LIN {X 0,Y 73.269,Z 1097.58,A -85,B 0,C 180,E1 32760.013,E2 32760.013} C_VEL
LIN {X 0,Y 72.331,Z 1070.54,A -85,B 0,C 180,E1 32774.928,E2 32774.928} C_VEL
LIN {X 0,Y 74.049,Z 1040.132,A -85,B 0,C 180,E1 32785.713,E2 32785.713} C_VEL
LIN {X 0,Y 75.716,Z 1012.125,A -85,B 0,C 180,E1 32791.765,E2 32791.765} C_VEL
LIN {X 0,Y 78.944,Z 1000.666,A -85,B 0,C 180,E1 32799.89,E2 32799.89} C_VEL
LIN {X 0,Y 85.957,Z 982.06,A -85,B 0,C 180,E1 32811.287,E2 32811.287} C_VEL
LIN {X 0,Y 92.075,Z 967.893,A -85,B 0,C 180,E1 32817.665,E2 32817.665} C_VEL
LIN {X 0,Y 97.491,Z 977.138,A -85,B 0,C 180,E1 32834.538,E2 32834.538} C_VEL
LIN {X 0,Y 99.424,Z 982.889,A -85,B 0,C 180,E1 32839.493,E2 32839.493} C_VEL
LIN {X 0,Y 102.891,Z 1004.981,A -85,B 0,C 180,E1 32851.504,E2 32851.504} C_VEL
LIN {X 0,Y 105.917,Z 1033.576,A -85,B 0,C 180,E1 32864.114,E2 32864.114} C_VEL
LIN {X 0,Y 108.13,Z 1063.069,A -85,B 0,C 180,E1 32876.43,E2 32876.43} C_VEL
LIN {X 0,Y 91.376,Z 1095.603,A -85,B 0,C 180,E1 32887.248,E2 32887.248} C_VEL
LIN {X 0,Y 75.131,Z 1127.363,A -85,B 0,C 180,E1 32906.405,E2 32906.405} C_VEL
LIN {X 0,Y 68.306,Z 1151.794,A -85,B 0,C 180,E1 32932.192,E2 32932.192} C_VEL
LIN {X 0,Y 69.608,Z 1165.233,A -85,B 0,C 180,E1 32952.524,E2 32952.524} C_VEL
LIN {X 0,Y 72.852,Z 1171.689,A -85,B 0,C 180,E1 32964.037,E2 32964.037} C_VEL
LIN {X 0,Y 74.21,Z 1174.974,A -85,B 0,C 180,E1 32972.734,E2 32972.734} C_VEL
LIN {X 0,Y 75.278,Z 1177.096,A -85,B 0,C 180,E1 32981.863,E2 32981.863} C_VEL
LIN {X 0,Y 76.32,Z 1177.928,A -85,B 0,C 180,E1 32984.944,E2 32984.944} C_VEL
LIN {X 0,Y 64.876,Z 1167.053,A -85,B 0,C 180,E1 33016.653,E2 33016.653} C_VEL
LIN {X 0,Y 64.458,Z 1162.406,A -85,B 0,C 180,E1 33026.759,E2 33026.759} C_VEL
LIN {X 0,Y 69.223,Z 1138.874,A -85,B 0,C 180,E1 33059.162,E2 33059.162} C_VEL
LIN {X 0,Y 77.507,Z 1130.596,A -85,B 0,C 180,E1 33067.478,E2 33067.478} C_VEL
LIN {X 0,Y 86.454,Z 1136.917,A -85,B 0,C 180,E1 33081.75,E2 33081.75} C_VEL
LIN {X 0,Y 88.495,Z 1137.46,A -85,B 0,C 180,E1 33084.935,E2 33084.935} C_VEL
LIN {X 0,Y 71.845,Z 1114.418,A -85,B 0,C 180,E1 33102.582,E2 33102.582} C_VEL
LIN {X 0,Y 65.942,Z 1089.767,A -85,B 0,C 180,E1 33120.835,E2 33120.835} C_VEL
LIN {X 0,Y 65.245,Z 1061.691,A -85,B 0,C 180,E1 33136.079,E2 33136.079} C_VEL
LIN {X 0,Y 66.642,Z 1034.04,A -85,B 0,C 180,E1 33146.198,E2 33146.198} C_VEL
LIN {X 0,Y 68.109,Z 1027.676,A -85,B 0,C 180,E1 33151.99,E2 33151.99} C_VEL
LIN {X 0,Y 72.601,Z 1016.135,A -85,B 0,C 180,E1 33156.945,E2 33156.945} C_VEL
LIN {X 0,Y 88.946,Z 978.744,A -85,B 0,C 180,E1 33179.557,E2 33179.557} C_VEL
LIN {X 0,Y 90.136,Z 977.435,A -85,B 0,C 180,E1 33181.585,E2 33181.585} C_VEL
LIN {X 0,Y 94.291,Z 984.5,A -85,B 0,C 180,E1 33194.097,E2 33194.097} C_VEL
LIN {X 0,Y 96.446,Z 998.943,A -85,B 0,C 180,E1 33203.737,E2 33203.737} C_VEL
LIN {X 0,Y 98.608,Z 1023.035,A -85,B 0,C 180,E1 33215.969,E2 33215.969} C_VEL
LIN {X 0,Y 100.362,Z 1052.462,A -85,B 0,C 180,E1 33229.311,E2 33229.311} C_VEL
LIN {X 0,Y 100.749,Z 1064.923,A -85,B 0,C 180,E1 33234.814,E2 33234.814} C_VEL
LIN {X 0,Y 80.54,Z 1101.135,A -85,B 0,C 180,E1 33248.2,E2 33248.2} C_VEL
LIN {X 0,Y 65.83,Z 1129.761,A -85,B 0,C 180,E1 33268.887,E2 33268.887} C_VEL
LIN {X 0,Y 60.684,Z 1152.02,A -85,B 0,C 180,E1 33296.409,E2 33296.409} C_VEL
LIN {X 0,Y 63.78,Z 1165.667,A -85,B 0,C 180,E1 33320.077,E2 33320.077} C_VEL
LIN {X 0,Y 75.278,Z 1177.096,A -85,B 0,C 180,E1 33341.863,E2 33341.863} C_VEL
LIN {X 0,Y 73.492,Z 1176.552,A -85,B 0,C 180,E1 33346.07,E2 33346.07} C_VEL
LIN {X 0,Y 61.63,Z 1169.7,A -85,B 0,C 180,E1 33356.97,E2 33356.97} C_VEL
LIN {X 0,Y 57.635,Z 1160.709,A -85,B 0,C 180,E1 33382.601,E2 33382.601} C_VEL
LIN {X 0,Y 60.537,Z 1138.156,A -85,B 0,C 180,E1 33418.076,E2 33418.076} C_VEL
LIN {X 0,Y 72.588,Z 1126.229,A -85,B 0,C 180,E1 33431.005,E2 33431.005} C_VEL
LIN {X 0,Y 80.021,Z 1131.328,A -85,B 0,C 180,E1 33443.585,E2 33443.585} C_VEL
LIN {X 0,Y 64.193,Z 1107.032,A -85,B 0,C 180,E1 33462.394,E2 33462.394} C_VEL
LIN {X 0,Y 58.753,Z 1082.208,A -85,B 0,C 180,E1 33480.937,E2 33480.937} C_VEL
LIN {X 0,Y 57.93,Z 1055.888,A -85,B 0,C 180,E1 33496.145,E2 33496.145} C_VEL
LIN {X 0,Y 59.201,Z 1047.428,A -85,B 0,C 180,E1 33505.556,E2 33505.556} C_VEL
LIN {X 0,Y 62.564,Z 1038.679,A -85,B 0,C 180,E1 33510.898,E2 33510.898} C_VEL
LIN {X 0,Y 66.244,Z 1028.558,A -85,B 0,C 180,E1 33518.87,E2 33518.87} C_VEL
LIN {X 0,Y 70.701,Z 1018.492,A -85,B 0,C 180,E1 33523.474,E2 33523.474} C_VEL
LIN {X 0,Y 87.345,Z 985.981,A -85,B 0,C 180,E1 33542.477,E2 33542.477} C_VEL
LIN {X 0,Y 90.25,Z 990.494,A -85,B 0,C 180,E1 33551.862,E2 33551.862} C_VEL
LIN {X 0,Y 91.426,Z 1000.781,A -85,B 0,C 180,E1 33559.484,E2 33559.484} C_VEL
LIN {X 0,Y 92.615,Z 1023.861,A -85,B 0,C 180,E1 33572.255,E2 33572.255} C_VEL
LIN {X 0,Y 93.504,Z 1052.595,A -85,B 0,C 180,E1 33586.339,E2 33586.339} C_VEL
LIN {X 0,Y 93.778,Z 1064.964,A -85,B 0,C 180,E1 33592.325,E2 33592.325} C_VEL
LIN {X 0,Y 74.007,Z 1099.068,A -85,B 0,C 180,E1 33605.219,E2 33605.219} C_VEL
LIN {X 0,Y 57.888,Z 1128.86,A -85,B 0,C 180,E1 33628.51,E2 33628.51} C_VEL
LIN {X 0,Y 53.268,Z 1149.848,A -85,B 0,C 180,E1 33657.947,E2 33657.947} C_VEL
LIN {X 0,Y 57.119,Z 1163.179,A -85,B 0,C 180,E1 33683.362,E2 33683.362} C_VEL
LIN {X 0,Y 67.223,Z 1172.897,A -85,B 0,C 180,E1 33702.869,E2 33702.869} C_VEL
LIN {X 0,Y 67.587,Z 1173.302,A -85,B 0,C 180,E1 33705.478,E2 33705.478} C_VEL
LIN {X 0,Y 61.63,Z 1169.7,A -85,B 0,C 180,E1 33716.97,E2 33716.97} C_VEL
LIN {X 0,Y 56.714,Z 1164.958,A -85,B 0,C 180,E1 33727.877,E2 33727.877} C_VEL
LIN {X 0,Y 49.623,Z 1154.018,A -85,B 0,C 180,E1 33747.821,E2 33747.821} C_VEL
LIN {X 0,Y 55.431,Z 1132.611,A -85,B 0,C 180,E1 33783.2,E2 33783.2} C_VEL
LIN {X 0,Y 67.962,Z 1121.517,A -85,B 0,C 180,E1 33794.648,E2 33794.648} C_VEL
LIN {X 0,Y 71.157,Z 1124.078,A -85,B 0,C 180,E1 33800.442,E2 33800.442} C_VEL
LIN {X 0,Y 71.261,Z 1123.721,A -85,B 0,C 180,E1 33802.452,E2 33802.452} C_VEL
LIN {X 0,Y 56.613,Z 1098.605,A -85,B 0,C 180,E1 33822.254,E2 33822.254} C_VEL
LIN {X 0,Y 51.874,Z 1079.167,A -85,B 0,C 180,E1 33837.931,E2 33837.931} C_VEL
LIN {X 0,Y 50.419,Z 1070.196,A -85,B 0,C 180,E1 33850.815,E2 33850.815} C_VEL
LIN {X 0,Y 52.781,Z 1060.211,A -85,B 0,C 180,E1 33861.06,E2 33861.06} C_VEL
LIN {X 0,Y 56.042,Z 1049.349,A -85,B 0,C 180,E1 33872.654,E2 33872.654} C_VEL
LIN {X 0,Y 59.41,Z 1041.697,A -85,B 0,C 180,E1 33877.872,E2 33877.872} C_VEL
LIN {X 0,Y 64.941,Z 1030.146,A -85,B 0,C 180,E1 33885.654,E2 33885.654} C_VEL
LIN {X 0,Y 70.113,Z 1019.904,A -85,B 0,C 180,E1 33890.545,E2 33890.545} C_VEL
LIN {X 0,Y 85.198,Z 994.192,A -85,B 0,C 180,E1 33905.357,E2 33905.357} C_VEL
LIN {X 0,Y 86.763,Z 999.12,A -85,B 0,C 180,E1 33912.164,E2 33912.164} C_VEL
LIN {X 0,Y 87.019,Z 1019.939,A -85,B 0,C 180,E1 33925.462,E2 33925.462} C_VEL
LIN {X 0,Y 86.841,Z 1046.993,A -85,B 0,C 180,E1 33939.931,E2 33939.931} C_VEL
LIN {X 0,Y 86.732,Z 1065.405,A -85,B 0,C 180,E1 33949.592,E2 33949.592} C_VEL
LIN {X 0,Y 66.137,Z 1099.464,A -85,B 0,C 180,E1 33963.197,E2 33963.197} C_VEL
LIN {X 0,Y 49.307,Z 1129.404,A -85,B 0,C 180,E1 33990.11,E2 33990.11} C_VEL
LIN {X 0,Y 46.044,Z 1148.807,A -85,B 0,C 180,E1 34022.331,E2 34022.331} C_VEL
LIN {X 0,Y 51.733,Z 1161.812,A -85,B 0,C 180,E1 34050.132,E2 34050.132} C_VEL
LIN {X 0,Y 59.063,Z 1168.261,A -85,B 0,C 180,E1 34063.449,E2 34063.449} C_VEL
LIN {X 0,Y 55.452,Z 1166.083,A -85,B 0,C 180,E1 34073.716,E2 34073.716} C_VEL
LIN {X 0,Y 50.452,Z 1157.108,A -85,B 0,C 180,E1 34101.541,E2 34101.541} C_VEL
LIN {X 0,Y 49.623,Z 1154.018,A -85,B 0,C 180,E1 34107.821,E2 34107.821} C_VEL
LIN {X 0,Y 46.659,Z 1146.453,A -85,B 0,C 180,E1 34120.097,E2 34120.097} C_VEL
LIN {X 0,Y 45.254,Z 1133.912,A -85,B 0,C 180,E1 34139.18,E2 34139.18} C_VEL
LIN {X 0,Y 46.03,Z 1132.614,A -85,B 0,C 180,E1 34141.155,E2 34141.155} C_VEL
LIN {X 0,Y 61.583,Z 1117.997,A -85,B 0,C 180,E1 34157.58,E2 34157.58} C_VEL
LIN {X 0,Y 63.777,Z 1116.677,A -85,B 0,C 180,E1 34158.781,E2 34158.781} C_VEL
LIN {X 0,Y 64.034,Z 1116.775,A -85,B 0,C 180,E1 34160.044,E2 34160.044} C_VEL
LIN {X 0,Y 58.379,Z 1109.531,A -85,B 0,C 180,E1 34165.532,E2 34165.532} C_VEL
LIN {X 0,Y 46.971,Z 1093.398,A -85,B 0,C 180,E1 34186.84,E2 34186.84} C_VEL
LIN {X 0,Y 45.464,Z 1083.478,A -85,B 0,C 180,E1 34200.552,E2 34200.552} C_VEL
LIN {X 0,Y 45.37,Z 1072.217,A -85,B 0,C 180,E1 34218.091,E2 34218.091} C_VEL
LIN {X 0,Y 48.213,Z 1063.415,A -85,B 0,C 180,E1 34228.232,E2 34228.232} C_VEL
LIN {X 0,Y 54.1,Z 1050.421,A -85,B 0,C 180,E1 34240.916,E2 34240.916} C_VEL
LIN {X 0,Y 64.463,Z 1031.664,A -85,B 0,C 180,E1 34252.58,E2 34252.58} C_VEL
LIN {X 0,Y 70.388,Z 1021.454,A -85,B 0,C 180,E1 34257.406,E2 34257.406} C_VEL
LIN {X 0,Y 81.875,Z 1004.023,A -85,B 0,C 180,E1 34267.37,E2 34267.37} C_VEL
LIN {X 0,Y 82.7,Z 1003.402,A -85,B 0,C 180,E1 34268.468,E2 34268.468} C_VEL
LIN {X 0,Y 81.933,Z 1022.116,A -85,B 0,C 180,E1 34281.289,E2 34281.289} C_VEL
LIN {X 0,Y 80.598,Z 1048.537,A -85,B 0,C 180,E1 34296.633,E2 34296.633} C_VEL
LIN {X 0,Y 79.874,Z 1065.624,A -85,B 0,C 180,E1 34306.312,E2 34306.312} C_VEL
LIN {X 0,Y 59.759,Z 1097.562,A -85,B 0,C 180,E1 34319.305,E2 34319.305} C_VEL
LIN {X 0,Y 41.409,Z 1128.292,A -85,B 0,C 180,E1 34349.857,E2 34349.857} C_VEL
LIN {X 0,Y 39.175,Z 1147.808,A -85,B 0,C 180,E1 34388.69,E2 34388.69} C_VEL
LIN {X 0,Y 50.045,Z 1162.565,A -85,B 0,C 180,E1 34423.182,E2 34423.182} C_VEL
LIN {X 0,Y 51.23,Z 1163.45,A -85,B 0,C 180,E1 34426.003,E2 34426.003} C_VEL
LIN {X 0,Y 44.027,Z 1155.114,A -85,B 0,C 180,E1 34455.264,E2 34455.264} C_VEL
LIN {X 0,Y 41.905,Z 1141.177,A -85,B 0,C 180,E1 34485.879,E2 34485.879} C_VEL
LIN {X 0,Y 46.03,Z 1132.614,A -85,B 0,C 180,E1 34501.155,E2 34501.155} C_VEL
LIN {X 0,Y 51.776,Z 1117.439,A -85,B 0,C 180,E1 34519.22,E2 34519.22} C_VEL
LIN {X 0,Y 52.783,Z 1116.6,A -85,B 0,C 180,E1 34519.963,E2 34519.963} C_VEL
LIN {X 0,Y 52.701,Z 1114.158,A -85,B 0,C 180,E1 34522.478,E2 34522.478} C_VEL
LIN {X 0,Y 40.236,Z 1097.736,A -85,B 0,C 180,E1 34547.208,E2 34547.208} C_VEL
LIN {X 0,Y 38.845,Z 1086.815,A -85,B 0,C 180,E1 34565.605,E2 34565.605} C_VEL
LIN {X 0,Y 41.251,Z 1073.821,A -85,B 0,C 180,E1 34587.276,E2 34587.276} C_VEL
LIN {X 0,Y 51.882,Z 1053.742,A -85,B 0,C 180,E1 34608.301,E2 34608.301} C_VEL
LIN {X 0,Y 64.406,Z 1033.964,A -85,B 0,C 180,E1 34619.298,E2 34619.298} C_VEL
LIN {X 0,Y 70.085,Z 1025.154,A -85,B 0,C 180,E1 34623.161,E2 34623.161} C_VEL
LIN {X 0,Y 78.268,Z 1014.107,A -85,B 0,C 180,E1 34629.629,E2 34629.629} C_VEL
LIN {X 0,Y 75.978,Z 1036.049,A -85,B 0,C 180,E1 34644.193,E2 34644.193} C_VEL
LIN {X 0,Y 73.393,Z 1064.578,A -85,B 0,C 180,E1 34661.774,E2 34661.774} C_VEL
LIN {X 0,Y 71.768,Z 1068.969,A -85,B 0,C 180,E1 34663.684,E2 34663.684} C_VEL
LIN {X 0,Y 48.037,Z 1103.645,A -85,B 0,C 180,E1 34680.072,E2 34680.072} C_VEL
LIN {X 0,Y 32.019,Z 1131.042,A -85,B 0,C 180,E1 34717.825,E2 34717.825} C_VEL
LIN {X 0,Y 33.455,Z 1147.512,A -85,B 0,C 180,E1 34759.772,E2 34759.772} C_VEL
LIN {X 0,Y 42.399,Z 1157.413,A -85,B 0,C 180,E1 34785.432,E2 34785.432} C_VEL
LIN {X 0,Y 38.023,Z 1152.822,A -85,B 0,C 180,E1 34806.804,E2 34806.804} C_VEL
LIN {X 0,Y 34.899,Z 1145.661,A -85,B 0,C 180,E1 34827.116,E2 34827.116} C_VEL
LIN {X 0,Y 42.009,Z 1126.064,A -85,B 0,C 180,E1 34869.242,E2 34869.242} C_VEL
LIN {X 0,Y 52.783,Z 1116.6,A -85,B 0,C 180,E1 34879.963,E2 34879.963} C_VEL
LIN {X 0,Y 51.395,Z 1113.671,A -85,B 0,C 180,E1 34883.224,E2 34883.224} C_VEL
LIN {X 0,Y 36.084,Z 1107.544,A -85,B 0,C 180,E1 34896.539,E2 34896.539} C_VEL
LIN {X 0,Y 35.699,Z 1107.001,A -85,B 0,C 180,E1 34897.623,E2 34897.623} C_VEL
LIN {X 0,Y 32.687,Z 1089.505,A -85,B 0,C 180,E1 34933.845,E2 34933.845} C_VEL
LIN {X 0,Y 38.353,Z 1075.343,A -85,B 0,C 180,E1 34958.016,E2 34958.016} C_VEL
LIN {X 0,Y 50.178,Z 1057.544,A -85,B 0,C 180,E1 34975.943,E2 34975.943} C_VEL
LIN {X 0,Y 65.017,Z 1036.397,A -85,B 0,C 180,E1 34985.916,E2 34985.916} C_VEL
LIN {X 0,Y 72.206,Z 1026.65,A -85,B 0,C 180,E1 34990.403,E2 34990.403} C_VEL
LIN {X 0,Y 73.006,Z 1025.797,A -85,B 0,C 180,E1 34991.067,E2 34991.067} C_VEL
LIN {X 0,Y 69.36,Z 1048.529,A -85,B 0,C 180,E1 35006.382,E2 35006.382} C_VEL
LIN {X 0,Y 66.702,Z 1067.325,A -85,B 0,C 180,E1 35018.844,E2 35018.844} C_VEL
LIN {X 0,Y 41.562,Z 1102.19,A -85,B 0,C 180,E1 35034.586,E2 35034.586} C_VEL
LIN {X 0,Y 24.042,Z 1130.282,A -85,B 0,C 180,E1 35081.554,E2 35081.554} C_VEL
LIN {X 0,Y 28.514,Z 1146.066,A -85,B 0,C 180,E1 35131.963,E2 35131.963} C_VEL
LIN {X 0,Y 33.734,Z 1151.068,A -85,B 0,C 180,E1 35146.21,E2 35146.21} C_VEL
LIN {X 0,Y 34.262,Z 1151.479,A -85,B 0,C 180,E1 35150.343,E2 35150.343} C_VEL
LIN {X 0,Y 30.015,Z 1146.152,A -85,B 0,C 180,E1 35171.929,E2 35171.929} C_VEL
LIN {X 0,Y 34.271,Z 1123.987,A -85,B 0,C 180,E1 35231.699,E2 35231.699} C_VEL
LIN {X 0,Y 42.454,Z 1116.366,A -85,B 0,C 180,E1 35241.976,E2 35241.976} C_VEL
LIN {X 0,Y 42.067,Z 1114.607,A -85,B 0,C 180,E1 35244.351,E2 35244.351} C_VEL
LIN {X 0,Y 35.699,Z 1107.001,A -85,B 0,C 180,E1 35257.623,E2 35257.623} C_VEL
LIN {X 0,Y 28.843,Z 1098.236,A -85,B 0,C 180,E1 35282.374,E2 35282.374} C_VEL
LIN {X 0,Y 28.812,Z 1089.021,A -85,B 0,C 180,E1 35312.75,E2 35312.75} C_VEL
LIN {X 0,Y 49.374,Z 1061.151,A -85,B 0,C 180,E1 35344.074,E2 35344.074} C_VEL
LIN {X 0,Y 65.343,Z 1040.222,A -85,B 0,C 180,E1 35352.14,E2 35352.14} C_VEL
LIN {X 0,Y 66.192,Z 1038.969,A -85,B 0,C 180,E1 35352.339,E2 35352.339} C_VEL
LIN {X 0,Y 66.097,Z 1041.687,A -85,B 0,C 180,E1 35355.293,E2 35355.293} C_VEL
LIN {X 0,Y 61.079,Z 1066.087,A -85,B 0,C 180,E1 35372.663,E2 35372.663} C_VEL
LIN {X 0,Y 57.823,Z 1071.773,A -85,B 0,C 180,E1 35374.725,E2 35374.725} C_VEL
LIN {X 0,Y 32.295,Z 1104.572,A -85,B 0,C 180,E1 35390.56,E2 35390.56} C_VEL
LIN {X 0,Y 16.295,Z 1129.964,A -85,B 0,C 180,E1 35451.378,E2 35451.378} C_VEL
LIN {X 0,Y 24.296,Z 1143.57,A -85,B 0,C 180,E1 35505.714,E2 35505.714} C_VEL
LIN {X 0,Y 25.874,Z 1144.891,A -85,B 0,C 180,E1 35509.553,E2 35509.553} C_VEL
LIN {X 0,Y 25.994,Z 1144.851,A -85,B 0,C 180,E1 35514.819,E2 35514.819} C_VEL
LIN {X 0,Y 28.171,Z 1120.39,A -85,B 0,C 180,E1 35598.109,E2 35598.109} C_VEL
LIN {X 0,Y 32.174,Z 1116.859,A -85,B 0,C 180,E1 35603.711,E2 35603.711} C_VEL
LIN {X 0,Y 30.671,Z 1113.321,A -85,B 0,C 180,E1 35610.517,E2 35610.517} C_VEL
LIN {X 0,Y 27.268,Z 1092.908,A -85,B 0,C 180,E1 35663.205,E2 35663.205} C_VEL
LIN {X 0,Y 28.812,Z 1089.021,A -85,B 0,C 180,E1 35672.75,E2 35672.75} C_VEL
LIN {X 0,Y 35.544,Z 1079.445,A -85,B 0,C 180,E1 35696.596,E2 35696.596} C_VEL
LIN {X 0,Y 44.353,Z 1070.714,A -85,B 0,C 180,E1 35709.683,E2 35709.683} C_VEL
LIN {X 0,Y 45.731,Z 1069.178,A -85,B 0,C 180,E1 35710.609,E2 35710.609} C_VEL
LIN {X 0,Y 56.628,Z 1056.346,A -85,B 0,C 180,E1 35715.374,E2 35715.374} C_VEL
LIN {X 0,Y 58.863,Z 1054.447,A -85,B 0,C 180,E1 35717.251,E2 35717.251} C_VEL
LIN {X 0,Y 55.414,Z 1067.461,A -85,B 0,C 180,E1 35727.239,E2 35727.239} C_VEL
LIN {X 0,Y 31.391,Z 1097.873,A -85,B 0,C 180,E1 35736.613,E2 35736.613} C_VEL
LIN {X 0,Y 9.111,Z 1125.263,A -85,B 0,C 180,E1 35804.447,E2 35804.447} C_VEL
LIN {X 0,Y 15.122,Z 1135.696,A -85,B 0,C 180,E1 35868.451,E2 35868.451} C_VEL
LIN {X 0,Y 16.665,Z 1136.873,A -85,B 0,C 180,E1 35877.525,E2 35877.525} C_VEL
LIN {X 0,Y 22.427,Z 1116.885,A -85,B 0,C 180,E1 35967.477,E2 35967.477} C_VEL
LIN {X 0,Y 20.407,Z 1111.748,A -85,B 0,C 180,E1 35982.937,E2 35982.937} C_VEL
LIN {X 0,Y 22.626,Z 1096.332,A -85,B 0,C 180,E1 36035.81,E2 36035.81} C_VEL
LIN {X 0,Y 45.731,Z 1069.178,A -85,B 0,C 180,E1 36070.609,E2 36070.609} C_VEL
LIN {X 0,Y 44.852,Z 1072.124,A -85,B 0,C 180,E1 36074.392,E2 36074.392} C_VEL
LIN {X 0,Y 41.744,Z 1077.469,A -85,B 0,C 180,E1 36077.222,E2 36077.222} C_VEL
LIN {X 0,Y 30.68,Z 1092.541,A -85,B 0,C 180,E1 36082.761,E2 36082.761} C_VEL
LIN {X 0,Y 26.509,Z 1097.161,A -85,B 0,C 180,E1 36083.846,E2 36083.846} C_VEL
LIN {X 0,Y 2.448,Z 1123.705,A -85,B 0,C 180,E1 36216.376,E2 36216.376} C_VEL
LIN {X 0,Y 5.22,Z 1126.269,A -85,B 0,C 180,E1 36243.143,E2 36243.143} C_VEL
LIN {X 0,Y 5.976,Z 1124.362,A -85,B 0,C 180,E1 36286.527,E2 36286.527} C_VEL
LIN {X 0,Y 13.057,Z 1116.834,A -85,B 0,C 180,E1 36336.165,E2 36336.165} C_VEL
LIN {X 0,Y 13.817,Z 1107.56,A -85,B 0,C 180,E1 36384.287,E2 36384.287} C_VEL
LIN {X 0,Y 32.953,Z 1086.113,A -85,B 0,C 180,E1 36431.646,E2 36431.646} C_VEL
LIN {X 0,Y 46.159,Z 1073.026,A -85,B 0,C 180,E1 36439.252,E2 36439.252} C_VEL
LIN {X 0,Y 45.095,Z 1075.295,A -85,B 0,C 180,E1 36440.903,E2 36440.903} C_VEL
LIN {X 0,Y 26.509,Z 1097.161,A -85,B 0,C 180,E1 36443.846,E2 36443.846} C_VEL
LIN {X 0,Y 25.96,Z 1098.539,A -85,B 0,C 180,E1 36443.92,E2 36443.92} C_VEL
LIN {X 0,Y 25.96,Z 1240.5,A -85,B 0,C 180,E1 36443.92,E2 36443.92} C_VEL
LIN {X 0,Y 25.96,Z 1240.5,A -85,B 0,C 180,E1 36443.92,E2 36443.92}

QRS_NEXT_CUT()
PTP {E1 36537.196,E2 36537.196}
PTP {X 0,Y 759.917,A -85,B 0,C 180,E1 36537.196,E2 36537.196,E3 0,E4 0,E5 0,E6 0}
QRS_SPEED_INIT()
LIN {X 0,Y 759.917,Z 1240.5,A -85,B 0,C 180,E1 36537.196,E2 36537.196,E3 0,E4 0,E5 0,E6 0} C_VEL
LIN {X 0,Y 759.917,Z 1178.221,A -85,B 0,C 180,E1 36537.196,E2 36537.196} C_VEL
LIN {X 0,Y 759.917,Z 1169.947,A -85,B 0,C 180,E1 36537.196,E2 36537.196} C_VEL
LIN {X 0,Y 759.916,Z 1167.96,A -85,B 0,C 180,E1 36537.062,E2 36537.062} C_VEL
LIN {X 0,Y 759.918,Z 1164.115,A -85,B 0,C 180,E1 36535.398,E2 36535.398} C_VEL
LIN {X 0,Y 759.917,Z 1158.554,A -85,B 0,C 180,E1 36533.732,E2 36533.732} C_VEL
LIN {X 0,Y 759.907,Z 1151.554,A -85,B 0,C 180,E1 36532.137,E2 36532.137} C_VEL
LIN {X 0,Y 759.915,Z 1143.032,A -85,B 0,C 180,E1 36530.612,E2 36530.612} C_VEL
LIN {X 0,Y 759.91,Z 1132.05,A -85,B 0,C 180,E1 36528.988,E2 36528.988} C_VEL
LIN {X 0,Y 759.905,Z 1120.121,A -85,B 0,C 180,E1 36527.509,E2 36527.509} C_VEL
LIN {X 0,Y 759.908,Z 1107.146,A -85,B 0,C 180,E1 36526.146,E2 36526.146} C_VEL
LIN {X 0,Y 759.913,Z 1092.503,A -85,B 0,C 180,E1 36524.823,E2 36524.823} C_VEL
LIN {X 0,Y 759.914,Z 1075.894,A -85,B 0,C 180,E1 36523.53,E2 36523.53} C_VEL
LIN {X 0,Y 759.919,Z 1058.852,A -85,B 0,C 180,E1 36522.386,E2 36522.386} C_VEL
LIN {X 0,Y 759.915,Z 1040.391,A -85,B 0,C 180,E1 36521.329,E2 36521.329} C_VEL
LIN {X 0,Y 759.917,Z 1021.211,A -85,B 0,C 180,E1 36520.398,E2 36520.398} C_VEL
LIN {X 0,Y 759.914,Z 1000.768,A -85,B 0,C 180,E1 36519.562,E2 36519.562} C_VEL
LIN {X 0,Y 759.918,Z 980.784,A -85,B 0,C 180,E1 36518.891,E2 36518.891} C_VEL
LIN {X 0,Y 759.914,Z 960.216,A -85,B 0,C 180,E1 36518.343,E2 36518.343} C_VEL
LIN {X 0,Y 759.906,Z 939.489,A -85,B 0,C 180,E1 36517.917,E2 36517.917} C_VEL
LIN {X 0,Y 759.907,Z 918.44,A -85,B 0,C 180,E1 36517.621,E2 36517.621} C_VEL
LIN {X 0,Y 759.917,Z 637.061,A -85,B 0,C 180,E1 36514.768,E2 36514.768} C_VEL
LIN {X 0,Y 759.907,Z 623.96,A -85,B 0,C 180,E1 36514.622,E2 36514.622} C_VEL
LIN {X 0,Y 759.883,Z 606.01,A -85,B 0,C 180,E1 36513.089,E2 36513.089} C_VEL
LIN {X 0,Y 759.884,Z 606.015,A -85,B 0,C 180,E1 36510.129,E2 36510.129} C_VEL
LIN {X 0,Y 759.822,Z 606.015,A -85,B 0,C 180,E1 36507.619,E2 36507.619} C_VEL
LIN {X 0,Y 759.857,Z 606.015,A -85,B 0,C 180,E1 36505.176,E2 36505.176} C_VEL
LIN {X 0,Y 759.885,Z 606.007,A -85,B 0,C 180,E1 36502.183,E2 36502.183} C_VEL
LIN {X 0,Y 759.903,Z 606.014,A -85,B 0,C 180,E1 36499.362,E2 36499.362} C_VEL
LIN {X 0,Y 759.911,Z 606.004,A -85,B 0,C 180,E1 36496.36,E2 36496.36} C_VEL
LIN {X 0,Y 759.874,Z 606.013,A -85,B 0,C 180,E1 36493.384,E2 36493.384} C_VEL
LIN {X 0,Y 759.831,Z 606.014,A -85,B 0,C 180,E1 36490.946,E2 36490.946} C_VEL
LIN {X 0,Y 759.895,Z 606.015,A -85,B 0,C 180,E1 36488.299,E2 36488.299} C_VEL
LIN {X 0,Y 759.859,Z 606.01,A -85,B 0,C 180,E1 36485.463,E2 36485.463} C_VEL
LIN {X 0,Y 759.905,Z 606.014,A -85,B 0,C 180,E1 36482.739,E2 36482.739} C_VEL
LIN {X 0,Y 759.909,Z 606.004,A -85,B 0,C 180,E1 36479.74,E2 36479.74} C_VEL
LIN {X 0,Y 759.885,Z 606.013,A -85,B 0,C 180,E1 36476.83,E2 36476.83} C_VEL
LIN {X 0,Y 759.851,Z 606.011,A -85,B 0,C 180,E1 36474.235,E2 36474.235} C_VEL
LIN {X 0,Y 759.897,Z 606.015,A -85,B 0,C 180,E1 36471.457,E2 36471.457} C_VEL
LIN {X 0,Y 759.84,Z 606.012,A -85,B 0,C 180,E1 36468.809,E2 36468.809} C_VEL
LIN {X 0,Y 759.895,Z 606.014,A -85,B 0,C 180,E1 36466.199,E2 36466.199} C_VEL
LIN {X 0,Y 759.906,Z 606.004,A -85,B 0,C 180,E1 36463.236,E2 36463.236} C_VEL
LIN {X 0,Y 759.898,Z 606.013,A -85,B 0,C 180,E1 36460.31,E2 36460.31} C_VEL
LIN {X 0,Y 759.874,Z 606.008,A -85,B 0,C 180,E1 36457.562,E2 36457.562} C_VEL
LIN {X 0,Y 759.859,Z 606.015,A -85,B 0,C 180,E1 36454.605,E2 36454.605} C_VEL
LIN {X 0,Y 759.824,Z 606.014,A -85,B 0,C 180,E1 36452.113,E2 36452.113} C_VEL
LIN {X 0,Y 759.898,Z 606.014,A -85,B 0,C 180,E1 36449.549,E2 36449.549} C_VEL
LIN {X 0,Y 759.889,Z 606.006,A -85,B 0,C 180,E1 36446.606,E2 36446.606} C_VEL
LIN {X 0,Y 759.902,Z 606.013,A -85,B 0,C 180,E1 36443.731,E2 36443.731} C_VEL
LIN {X 0,Y 759.905,Z 606.005,A -85,B 0,C 180,E1 36440.84,E2 36440.84} C_VEL
LIN {X 0,Y 759.857,Z 606.014,A -85,B 0,C 180,E1 36437.924,E2 36437.924} C_VEL
LIN {X 0,Y 759.82,Z 606.015,A -85,B 0,C 180,E1 36435.522,E2 36435.522} C_VEL
LIN {X 0,Y 759.895,Z 606.015,A -85,B 0,C 180,E1 36432.938,E2 36432.938} C_VEL
LIN {X 0,Y 759.878,Z 606.008,A -85,B 0,C 180,E1 36430.075,E2 36430.075} C_VEL
LIN {X 0,Y 759.911,Z 606.015,A -85,B 0,C 180,E1 36427.243,E2 36427.243} C_VEL
LIN {X 0,Y 759.917,Z 606.004,A -85,B 0,C 180,E1 36424.267,E2 36424.267} C_VEL
LIN {X 0,Y 759.868,Z 606.013,A -85,B 0,C 180,E1 36421.359,E2 36421.359} C_VEL
LIN {X 0,Y 759.831,Z 606.014,A -85,B 0,C 180,E1 36418.86,E2 36418.86} C_VEL
LIN {X 0,Y 759.917,Z 606.013,A -85,B 0,C 180,E1 36416.092,E2 36416.092} C_VEL
LIN {X 0,Y 759.856,Z 606.011,A -85,B 0,C 180,E1 36413.317,E2 36413.317} C_VEL
LIN {X 0,Y 759.909,Z 606.016,A -85,B 0,C 180,E1 36410.64,E2 36410.64} C_VEL
LIN {X 0,Y 759.908,Z 606.005,A -85,B 0,C 180,E1 36407.683,E2 36407.683} C_VEL
LIN {X 0,Y 759.882,Z 606.013,A -85,B 0,C 180,E1 36404.829,E2 36404.829} C_VEL
LIN {X 0,Y 759.852,Z 606.012,A -85,B 0,C 180,E1 36402.199,E2 36402.199} C_VEL
LIN {X 0,Y 759.87,Z 606.015,A -85,B 0,C 180,E1 36399.313,E2 36399.313} C_VEL
LIN {X 0,Y 759.844,Z 606.149,A -85,B 0,C 180,E1 36396.855,E2 36396.855} C_VEL
LIN {X 0,Y 759.916,Z 641.009,A -85,B 0,C 180,E1 36394.454,E2 36394.454} C_VEL
LIN {X 0,Y 759.906,Z 680.943,A -85,B 0,C 180,E1 36391.647,E2 36391.647} C_VEL
LIN {X 0,Y 759.874,Z 720.551,A -85,B 0,C 180,E1 36388.914,E2 36388.914} C_VEL
LIN {X 0,Y 759.871,Z 758.704,A -85,B 0,C 180,E1 36386.322,E2 36386.322} C_VEL
LIN {X 0,Y 759.909,Z 799.658,A -85,B 0,C 180,E1 36383.576,E2 36383.576} C_VEL
LIN {X 0,Y 759.901,Z 815.283,A -85,B 0,C 180,E1 36382.551,E2 36382.551} C_VEL
LIN {X 0,Y 759.913,Z 956.141,A -85,B 0,C 180,E1 36381.201,E2 36381.201} C_VEL
LIN {X 0,Y 759.899,Z 972.65,A -85,B 0,C 180,E1 36380.901,E2 36380.901} C_VEL
LIN {X 0,Y 759.9,Z 988.331,A -85,B 0,C 180,E1 36380.475,E2 36380.475} C_VEL
LIN {X 0,Y 759.896,Z 1003.054,A -85,B 0,C 180,E1 36379.923,E2 36379.923} C_VEL
LIN {X 0,Y 759.919,Z 1017.2,A -85,B 0,C 180,E1 36379.243,E2 36379.243} C_VEL
LIN {X 0,Y 759.919,Z 1029.687,A -85,B 0,C 180,E1 36378.486,E2 36378.486} C_VEL
LIN {X 0,Y 759.919,Z 1042.257,A -85,B 0,C 180,E1 36377.534,E2 36377.534} C_VEL
LIN {X 0,Y 759.91,Z 1052.212,A -85,B 0,C 180,E1 36376.588,E2 36376.588} C_VEL
LIN {X 0,Y 759.919,Z 1061.416,A -85,B 0,C 180,E1 36375.49,E2 36375.49} C_VEL
LIN {X 0,Y 759.915,Z 1068.501,A -85,B 0,C 180,E1 36374.398,E2 36374.398} C_VEL
LIN {X 0,Y 759.915,Z 1074.259,A -85,B 0,C 180,E1 36373.182,E2 36373.182} C_VEL
LIN {X 0,Y 759.916,Z 1078.04,A -85,B 0,C 180,E1 36371.997,E2 36371.997} C_VEL
LIN {X 0,Y 759.919,Z 1080.084,A -85,B 0,C 180,E1 36370.767,E2 36370.767} C_VEL
LIN {X 0,Y 759.917,Z 1080.385,A -85,B 0,C 180,E1 36369.541,E2 36369.541} C_VEL
LIN {X 0,Y 759.917,Z 1078.905,A -85,B 0,C 180,E1 36368.32,E2 36368.32} C_VEL
LIN {X 0,Y 759.918,Z 1075.641,A -85,B 0,C 180,E1 36367.103,E2 36367.103} C_VEL
LIN {X 0,Y 759.915,Z 1070.571,A -85,B 0,C 180,E1 36365.899,E2 36365.899} C_VEL
LIN {X 0,Y 759.915,Z 1063.767,A -85,B 0,C 180,E1 36364.753,E2 36364.753} C_VEL
LIN {X 0,Y 759.916,Z 1055.619,A -85,B 0,C 180,E1 36363.695,E2 36363.695} C_VEL
LIN {X 0,Y 759.917,Z 1046.049,A -85,B 0,C 180,E1 36362.713,E2 36362.713} C_VEL
LIN {X 0,Y 759.919,Z 1033.587,A -85,B 0,C 180,E1 36361.695,E2 36361.695} C_VEL
LIN {X 0,Y 759.919,Z 1020.711,A -85,B 0,C 180,E1 36360.865,E2 36360.865} C_VEL
LIN {X 0,Y 759.877,Z 1006.804,A -85,B 0,C 180,E1 36360.149,E2 36360.149} C_VEL
LIN {X 0,Y 759.88,Z 992.682,A -85,B 0,C 180,E1 36359.584,E2 36359.584} C_VEL
LIN {X 0,Y 759.918,Z 976.272,A -85,B 0,C 180,E1 36359.094,E2 36359.094} C_VEL
LIN {X 0,Y 759.913,Z 960.492,A -85,B 0,C 180,E1 36358.773,E2 36358.773} C_VEL
LIN {X 0,Y 759.916,Z 938.781,A -85,B 0,C 180,E1 36358.528,E2 36358.528} C_VEL
LIN {X 0,Y 759.912,Z 814.794,A -85,B 0,C 180,E1 36357.34,E2 36357.34} C_VEL
LIN {X 0,Y 759.915,Z 771.469,A -85,B 0,C 180,E1 36354.449,E2 36354.449} C_VEL
LIN {X 0,Y 759.854,Z 731.624,A -85,B 0,C 180,E1 36351.752,E2 36351.752} C_VEL
LIN {X 0,Y 759.873,Z 694.879,A -85,B 0,C 180,E1 36349.229,E2 36349.229} C_VEL
LIN {X 0,Y 759.916,Z 655.136,A -85,B 0,C 180,E1 36346.454,E2 36346.454} C_VEL
LIN {X 0,Y 759.914,Z 623.555,A -85,B 0,C 180,E1 36344.272,E2 36344.272} C_VEL
LIN {X 0,Y 759.872,Z 606.016,A -85,B 0,C 180,E1 36343.132,E2 36343.132} C_VEL
LIN {X 0,Y 759.869,Z 606.015,A -85,B 0,C 180,E1 36340.473,E2 36340.473} C_VEL
LIN {X 0,Y 759.904,Z 606.011,A -85,B 0,C 180,E1 36337.567,E2 36337.567} C_VEL
LIN {X 0,Y 759.875,Z 606.015,A -85,B 0,C 180,E1 36334.763,E2 36334.763} C_VEL
LIN {X 0,Y 759.889,Z 606.013,A -85,B 0,C 180,E1 36331.981,E2 36331.981} C_VEL
LIN {X 0,Y 759.904,Z 606.013,A -85,B 0,C 180,E1 36329.079,E2 36329.079} C_VEL
LIN {X 0,Y 759.892,Z 606.015,A -85,B 0,C 180,E1 36326.261,E2 36326.261} C_VEL
LIN {X 0,Y 759.916,Z 606.014,A -85,B 0,C 180,E1 36323.379,E2 36323.379} C_VEL
LIN {X 0,Y 759.909,Z 606.015,A -85,B 0,C 180,E1 36320.442,E2 36320.442} C_VEL
LIN {X 0,Y 759.914,Z 606.012,A -85,B 0,C 180,E1 36317.545,E2 36317.545} C_VEL
LIN {X 0,Y 759.885,Z 606.015,A -85,B 0,C 180,E1 36314.719,E2 36314.719} C_VEL
LIN {X 0,Y 759.895,Z 606.014,A -85,B 0,C 180,E1 36311.945,E2 36311.945} C_VEL
LIN {X 0,Y 759.918,Z 606.01,A -85,B 0,C 180,E1 36309.067,E2 36309.067} C_VEL
LIN {X 0,Y 759.87,Z 606.015,A -85,B 0,C 180,E1 36306.214,E2 36306.214} C_VEL
LIN {X 0,Y 759.893,Z 606.013,A -85,B 0,C 180,E1 36303.547,E2 36303.547} C_VEL
LIN {X 0,Y 759.915,Z 606.055,A -85,B 0,C 180,E1 36300.829,E2 36300.829} C_VEL
LIN {X 0,Y 759.902,Z 645.059,A -85,B 0,C 180,E1 36298.003,E2 36298.003} C_VEL
LIN {X 0,Y 759.853,Z 681.337,A -85,B 0,C 180,E1 36295.442,E2 36295.442} C_VEL
LIN {X 0,Y 759.861,Z 682.915,A -85,B 0,C 180,E1 36295.333,E2 36295.333} C_VEL
LIN {X 0,Y 759.911,Z 970.476,A -85,B 0,C 180,E1 36292.42,E2 36292.42} C_VEL
LIN {X 0,Y 759.904,Z 993.716,A -85,B 0,C 180,E1 36292.129,E2 36292.129} C_VEL
LIN {X 0,Y 759.916,Z 1014.182,A -85,B 0,C 180,E1 36291.753,E2 36291.753} C_VEL
LIN {X 0,Y 759.908,Z 1034.921,A -85,B 0,C 180,E1 36291.232,E2 36291.232} C_VEL
LIN {X 0,Y 759.917,Z 1055.932,A -85,B 0,C 180,E1 36290.566,E2 36290.566} C_VEL
LIN {X 0,Y 759.919,Z 1075.437,A -85,B 0,C 180,E1 36289.815,E2 36289.815} C_VEL
LIN {X 0,Y 759.916,Z 1094.348,A -85,B 0,C 180,E1 36288.934,E2 36288.934} C_VEL
LIN {X 0,Y 759.916,Z 1113.456,A -85,B 0,C 180,E1 36287.891,E2 36287.891} C_VEL
LIN {X 0,Y 759.914,Z 1130.834,A -85,B 0,C 180,E1 36286.786,E2 36286.786} C_VEL
LIN {X 0,Y 759.911,Z 1147.732,A -85,B 0,C 180,E1 36285.53,E2 36285.53} C_VEL
LIN {X 0,Y 759.915,Z 1162.571,A -85,B 0,C 180,E1 36284.243,E2 36284.243} C_VEL
LIN {X 0,Y 759.913,Z 1176.559,A -85,B 0,C 180,E1 36282.836,E2 36282.836} C_VEL
LIN {X 0,Y 759.91,Z 1188.932,A -85,B 0,C 180,E1 36281.382,E2 36281.382} C_VEL
LIN {X 0,Y 759.907,Z 1199.365,A -85,B 0,C 180,E1 36279.924,E2 36279.924} C_VEL
LIN {X 0,Y 759.914,Z 1208.478,A -85,B 0,C 180,E1 36278.397,E2 36278.397} C_VEL
LIN {X 0,Y 759.902,Z 1215.939,A -85,B 0,C 180,E1 36276.876,E2 36276.876} C_VEL
LIN {X 0,Y 759.912,Z 1221.908,A -85,B 0,C 180,E1 36275.284,E2 36275.284} C_VEL
LIN {X 0,Y 759.912,Z 1226.624,A -85,B 0,C 180,E1 36273.544,E2 36273.544} C_VEL
LIN {X 0,Y 759.918,Z 1229.416,A -85,B 0,C 180,E1 36271.884,E2 36271.884} C_VEL
LIN {X 0,Y 759.903,Z 1230.44,A -85,B 0,C 180,E1 36270.225,E2 36270.225} C_VEL
LIN {X 0,Y 759.898,Z 1229.813,A -85,B 0,C 180,E1 36268.566,E2 36268.566} C_VEL
LIN {X 0,Y 759.898,Z 1227.724,A -85,B 0,C 180,E1 36266.982,E2 36266.982} C_VEL
LIN {X 0,Y 759.906,Z 1223.985,A -85,B 0,C 180,E1 36265.395,E2 36265.395} C_VEL
LIN {X 0,Y 759.917,Z 1218.363,A -85,B 0,C 180,E1 36263.729,E2 36263.729} C_VEL
LIN {X 0,Y 759.909,Z 1211.309,A -85,B 0,C 180,E1 36262.134,E2 36262.134} C_VEL
LIN {X 0,Y 759.902,Z 1202.744,A -85,B 0,C 180,E1 36260.609,E2 36260.609} C_VEL
LIN {X 0,Y 759.902,Z 1192.38,A -85,B 0,C 180,E1 36259.077,E2 36259.077} C_VEL
LIN {X 0,Y 759.915,Z 1180.667,A -85,B 0,C 180,E1 36257.614,E2 36257.614} C_VEL
LIN {X 0,Y 759.907,Z 1167.082,A -85,B 0,C 180,E1 36256.185,E2 36256.185} C_VEL
LIN {X 0,Y 759.909,Z 1152.859,A -85,B 0,C 180,E1 36254.898,E2 36254.898} C_VEL
LIN {X 0,Y 759.914,Z 1136.873,A -85,B 0,C 180,E1 36253.645,E2 36253.645} C_VEL
LIN {X 0,Y 759.915,Z 1120.016,A -85,B 0,C 180,E1 36252.502,E2 36252.502} C_VEL
LIN {X 0,Y 759.919,Z 1102.173,A -85,B 0,C 180,E1 36251.472,E2 36251.472} C_VEL
LIN {X 0,Y 759.919,Z 1082.811,A -85,B 0,C 180,E1 36250.515,E2 36250.515} C_VEL
LIN {X 0,Y 759.918,Z 1063.594,A -85,B 0,C 180,E1 36249.709,E2 36249.709} C_VEL
LIN {X 0,Y 759.915,Z 1043.704,A -85,B 0,C 180,E1 36249.028,E2 36249.028} C_VEL
LIN {X 0,Y 759.907,Z 1021.622,A -85,B 0,C 180,E1 36248.421,E2 36248.421} C_VEL
LIN {X 0,Y 759.906,Z 1000.31,A -85,B 0,C 180,E1 36247.975,E2 36247.975} C_VEL
LIN {X 0,Y 759.907,Z 978.848,A -85,B 0,C 180,E1 36247.671,E2 36247.671} C_VEL
LIN {X 0,Y 759.865,Z 687.972,A -85,B 0,C 180,E1 36244.719,E2 36244.719} C_VEL
LIN {X 0,Y 759.86,Z 682.778,A -85,B 0,C 180,E1 36244.659,E2 36244.659} C_VEL
LIN {X 0,Y 759.895,Z 646.043,A -85,B 0,C 180,E1 36242.067,E2 36242.067} C_VEL
LIN {X 0,Y 759.912,Z 606.62,A -85,B 0,C 180,E1 36239.213,E2 36239.213} C_VEL
LIN {X 0,Y 759.914,Z 606.005,A -85,B 0,C 180,E1 36239.147,E2 36239.147} C_VEL
LIN {X 0,Y 759.904,Z 606.014,A -85,B 0,C 180,E1 36236.088,E2 36236.088} C_VEL
LIN {X 0,Y 759.892,Z 606.004,A -85,B 0,C 180,E1 36233.222,E2 36233.222} C_VEL
LIN {X 0,Y 759.907,Z 606.012,A -85,B 0,C 180,E1 36230.332,E2 36230.332} C_VEL
LIN {X 0,Y 759.87,Z 606.009,A -85,B 0,C 180,E1 36227.542,E2 36227.542} C_VEL
LIN {X 0,Y 759.907,Z 606.003,A -85,B 0,C 180,E1 36224.828,E2 36224.828} C_VEL
LIN {X 0,Y 759.89,Z 606.013,A -85,B 0,C 180,E1 36221.847,E2 36221.847} C_VEL
LIN {X 0,Y 759.859,Z 606.008,A -85,B 0,C 180,E1 36219.171,E2 36219.171} C_VEL
LIN {X 0,Y 759.911,Z 606.005,A -85,B 0,C 180,E1 36216.49,E2 36216.49} C_VEL
LIN {X 0,Y 759.863,Z 606.013,A -85,B 0,C 180,E1 36213.552,E2 36213.552} C_VEL
LIN {X 0,Y 759.845,Z 606.01,A -85,B 0,C 180,E1 36211.055,E2 36211.055} C_VEL
LIN {X 0,Y 759.904,Z 606.007,A -85,B 0,C 180,E1 36208.361,E2 36208.361} C_VEL
LIN {X 0,Y 759.847,Z 606.196,A -85,B 0,C 180,E1 36206.79,E2 36206.79} C_VEL
LIN {X 0,Y 759.869,Z 624.326,A -85,B 0,C 180,E1 36205.274,E2 36205.274} C_VEL
LIN {X 0,Y 759.91,Z 883.32,A -85,B 0,C 180,E1 36202.647,E2 36202.647} C_VEL
LIN {X 0,Y 759.918,Z 927.91,A -85,B 0,C 180,E1 36202.174,E2 36202.174} C_VEL
LIN {X 0,Y 759.917,Z 949.492,A -85,B 0,C 180,E1 36201.802,E2 36201.802} C_VEL
LIN {X 0,Y 759.906,Z 970.989,A -85,B 0,C 180,E1 36201.296,E2 36201.296} C_VEL
LIN {X 0,Y 759.903,Z 991.383,A -85,B 0,C 180,E1 36200.684,E2 36200.684} C_VEL
LIN {X 0,Y 759.918,Z 1011.559,A -85,B 0,C 180,E1 36199.926,E2 36199.926} C_VEL
LIN {X 0,Y 759.915,Z 1031.99,A -85,B 0,C 180,E1 36199.007,E2 36199.007} C_VEL
LIN {X 0,Y 759.917,Z 1050.681,A -85,B 0,C 180,E1 36198.013,E2 36198.013} C_VEL
LIN {X 0,Y 759.915,Z 1068.984,A -85,B 0,C 180,E1 36196.867,E2 36196.867} C_VEL
LIN {X 0,Y 759.917,Z 1085.602,A -85,B 0,C 180,E1 36195.65,E2 36195.65} C_VEL
LIN {X 0,Y 759.908,Z 1101.204,A -85,B 0,C 180,E1 36194.323,E2 36194.323} C_VEL
LIN {X 0,Y 759.905,Z 1115.317,A -85,B 0,C 180,E1 36192.927,E2 36192.927} C_VEL
LIN {X 0,Y 759.916,Z 1127.985,A -85,B 0,C 180,E1 36191.461,E2 36191.461} C_VEL
LIN {X 0,Y 759.901,Z 1138.526,A -85,B 0,C 180,E1 36190.004,E2 36190.004} C_VEL
LIN {X 0,Y 759.899,Z 1148.224,A -85,B 0,C 180,E1 36188.4,E2 36188.4} C_VEL
LIN {X 0,Y 759.904,Z 1155.721,A -85,B 0,C 180,E1 36186.879,E2 36186.879} C_VEL
LIN {X 0,Y 759.919,Z 1161.749,A -85,B 0,C 180,E1 36185.286,E2 36185.286} C_VEL
LIN {X 0,Y 759.915,Z 1166.367,A -85,B 0,C 180,E1 36183.623,E2 36183.623} C_VEL
LIN {X 0,Y 759.898,Z 1169.16,A -85,B 0,C 180,E1 36182.038,E2 36182.038} C_VEL
LIN {X 0,Y 759.898,Z 1170.36,A -85,B 0,C 180,E1 36180.454,E2 36180.454} C_VEL
LIN {X 0,Y 759.908,Z 1170.054,A -85,B 0,C 180,E1 36178.795,E2 36178.795} C_VEL
LIN {X 0,Y 759.916,Z 1168.07,A -85,B 0,C 180,E1 36177.136,E2 36177.136} C_VEL
LIN {X 0,Y 759.916,Z 1167.96,A -85,B 0,C 180,E1 36177.062,E2 36177.062} C_VEL
LIN {X 0,Y 758.93,Z 1166.935,A -85,B 0,C 180,E1 36176.487,E2 36176.487} C_VEL
LIN {X 0,Y 752.574,Z 1162.946,A -85,B 0,C 180,E1 36174.932,E2 36174.932} C_VEL
LIN {X 0,Y 751.912,Z 1161.465,A -85,B 0,C 180,E1 36174.48,E2 36174.48} C_VEL
LIN {X 0,Y 751.922,Z 1155.095,A -85,B 0,C 180,E1 36172.821,E2 36172.821} C_VEL
LIN {X 0,Y 751.923,Z 1147.503,A -85,B 0,C 180,E1 36171.283,E2 36171.283} C_VEL
LIN {X 0,Y 751.93,Z 1138.12,A -85,B 0,C 180,E1 36169.738,E2 36169.738} C_VEL
LIN {X 0,Y 751.955,Z 1127.485,A -85,B 0,C 180,E1 36168.263,E2 36168.263} C_VEL
LIN {X 0,Y 751.978,Z 1114.755,A -85,B 0,C 180,E1 36166.781,E2 36166.781} C_VEL
LIN {X 0,Y 752.017,Z 1100.524,A -85,B 0,C 180,E1 36165.369,E2 36165.369} C_VEL
LIN {X 0,Y 752.07,Z 1084.379,A -85,B 0,C 180,E1 36163.996,E2 36163.996} C_VEL
LIN {X 0,Y 752.125,Z 1067.397,A -85,B 0,C 180,E1 36162.757,E2 36162.757} C_VEL
LIN {X 0,Y 752.181,Z 1049.556,A -85,B 0,C 180,E1 36161.638,E2 36161.638} C_VEL
LIN {X 0,Y 752.237,Z 1030.656,A -85,B 0,C 180,E1 36160.634,E2 36160.634} C_VEL
LIN {X 0,Y 752.308,Z 1010.89,A -85,B 0,C 180,E1 36159.745,E2 36159.745} C_VEL
LIN {X 0,Y 752.361,Z 990.315,A -85,B 0,C 180,E1 36158.974,E2 36158.974} C_VEL
LIN {X 0,Y 752.406,Z 969.963,A -85,B 0,C 180,E1 36158.362,E2 36158.362} C_VEL
LIN {X 0,Y 752.462,Z 947.798,A -85,B 0,C 180,E1 36157.847,E2 36157.847} C_VEL
LIN {X 0,Y 752.493,Z 926.435,A -85,B 0,C 180,E1 36157.485,E2 36157.485} C_VEL
LIN {X 0,Y 752.572,Z 806.297,A -85,B 0,C 180,E1 36156.245,E2 36156.245} C_VEL
LIN {X 0,Y 752.475,Z 625.048,A -85,B 0,C 180,E1 36154.377,E2 36154.377} C_VEL
LIN {X 0,Y 752.283,Z 623.71,A -85,B 0,C 180,E1 36154.325,E2 36154.325} C_VEL
LIN {X 0,Y 752.095,Z 607.789,A -85,B 0,C 180,E1 36152.958,E2 36152.958} C_VEL
LIN {X 0,Y 751.966,Z 607,A -85,B 0,C 180,E1 36152.868,E2 36152.868} C_VEL
LIN {X 0,Y 751.918,Z 607.004,A -85,B 0,C 180,E1 36149.915,E2 36149.915} C_VEL
LIN {X 0,Y 751.883,Z 607.005,A -85,B 0,C 180,E1 36147.472,E2 36147.472} C_VEL
LIN {X 0,Y 751.977,Z 607.004,A -85,B 0,C 180,E1 36144.757,E2 36144.757} C_VEL
LIN {X 0,Y 751.93,Z 606.998,A -85,B 0,C 180,E1 36141.905,E2 36141.905} C_VEL
LIN {X 0,Y 751.971,Z 607.002,A -85,B 0,C 180,E1 36139.144,E2 36139.144} C_VEL
LIN {X 0,Y 751.977,Z 606.993,A -85,B 0,C 180,E1 36136.222,E2 36136.222} C_VEL
LIN {X 0,Y 751.929,Z 607.002,A -85,B 0,C 180,E1 36133.327,E2 36133.327} C_VEL
LIN {X 0,Y 751.896,Z 607.003,A -85,B 0,C 180,E1 36130.832,E2 36130.832} C_VEL
LIN {X 0,Y 751.969,Z 607.001,A -85,B 0,C 180,E1 36128,E2 36128} C_VEL
LIN {X 0,Y 751.915,Z 607,A -85,B 0,C 180,E1 36125.249,E2 36125.249} C_VEL
LIN {X 0,Y 751.974,Z 607.002,A -85,B 0,C 180,E1 36122.545,E2 36122.545} C_VEL
LIN {X 0,Y 751.964,Z 606.995,A -85,B 0,C 180,E1 36119.59,E2 36119.59} C_VEL
LIN {X 0,Y 751.943,Z 607.002,A -85,B 0,C 180,E1 36116.795,E2 36116.795} C_VEL
LIN {X 0,Y 751.916,Z 607,A -85,B 0,C 180,E1 36114.179,E2 36114.179} C_VEL
LIN {X 0,Y 751.93,Z 607.004,A -85,B 0,C 180,E1 36111.287,E2 36111.287} C_VEL
LIN {X 0,Y 751.901,Z 607.002,A -85,B 0,C 180,E1 36108.693,E2 36108.693} C_VEL
LIN {X 0,Y 751.976,Z 607.003,A -85,B 0,C 180,E1 36105.977,E2 36105.977} C_VEL
LIN {X 0,Y 751.955,Z 606.995,A -85,B 0,C 180,E1 36103.066,E2 36103.066} C_VEL
LIN {X 0,Y 751.954,Z 607.002,A -85,B 0,C 180,E1 36100.265,E2 36100.265} C_VEL
LIN {X 0,Y 751.942,Z 606.997,A -85,B 0,C 180,E1 36097.489,E2 36097.489} C_VEL
LIN {X 0,Y 751.907,Z 607.004,A -85,B 0,C 180,E1 36094.501,E2 36094.501} C_VEL
LIN {X 0,Y 751.887,Z 607.003,A -85,B 0,C 180,E1 36092.059,E2 36092.059} C_VEL
LIN {X 0,Y 751.974,Z 607.004,A -85,B 0,C 180,E1 36089.392,E2 36089.392} C_VEL
LIN {X 0,Y 751.944,Z 606.996,A -85,B 0,C 180,E1 36086.494,E2 36086.494} C_VEL
LIN {X 0,Y 751.964,Z 607.002,A -85,B 0,C 180,E1 36083.741,E2 36083.741} C_VEL
LIN {X 0,Y 751.96,Z 606.995,A -85,B 0,C 180,E1 36080.897,E2 36080.897} C_VEL
LIN {X 0,Y 751.92,Z 607.003,A -85,B 0,C 180,E1 36077.951,E2 36077.951} C_VEL
LIN {X 0,Y 751.882,Z 607.004,A -85,B 0,C 180,E1 36075.523,E2 36075.523} C_VEL
LIN {X 0,Y 751.961,Z 607.004,A -85,B 0,C 180,E1 36072.912,E2 36072.912} C_VEL
LIN {X 0,Y 751.936,Z 606.997,A -85,B 0,C 180,E1 36070.018,E2 36070.018} C_VEL
LIN {X 0,Y 751.972,Z 607.004,A -85,B 0,C 180,E1 36067.237,E2 36067.237} C_VEL
LIN {X 0,Y 751.974,Z 606.993,A -85,B 0,C 180,E1 36064.313,E2 36064.313} C_VEL
LIN {X 0,Y 751.93,Z 607.002,A -85,B 0,C 180,E1 36061.354,E2 36061.354} C_VEL
LIN {X 0,Y 751.893,Z 607.003,A -85,B 0,C 180,E1 36058.85,E2 36058.85} C_VEL
LIN {X 0,Y 751.974,Z 607.001,A -85,B 0,C 180,E1 36056.052,E2 36056.052} C_VEL
LIN {X 0,Y 751.917,Z 607,A -85,B 0,C 180,E1 36053.246,E2 36053.246} C_VEL
LIN {X 0,Y 751.97,Z 607.002,A -85,B 0,C 180,E1 36050.538,E2 36050.538} C_VEL
LIN {X 0,Y 751.965,Z 606.995,A -85,B 0,C 180,E1 36047.613,E2 36047.613} C_VEL
LIN {X 0,Y 751.938,Z 607.002,A -85,B 0,C 180,E1 36044.76,E2 36044.76} C_VEL
LIN {X 0,Y 751.914,Z 607.001,A -85,B 0,C 180,E1 36042.183,E2 36042.183} C_VEL
LIN {X 0,Y 751.924,Z 607.005,A -85,B 0,C 180,E1 36039.267,E2 36039.267} C_VEL
LIN {X 0,Y 751.936,Z 607.171,A -85,B 0,C 180,E1 36037.025,E2 36037.025} C_VEL
LIN {X 0,Y 752.222,Z 630.531,A -85,B 0,C 180,E1 36035.416,E2 36035.416} C_VEL
LIN {X 0,Y 752.251,Z 670.496,A -85,B 0,C 180,E1 36032.618,E2 36032.618} C_VEL
LIN {X 0,Y 752.176,Z 710.534,A -85,B 0,C 180,E1 36029.81,E2 36029.81} C_VEL
LIN {X 0,Y 752.077,Z 751.269,A -85,B 0,C 180,E1 36027.004,E2 36027.004} C_VEL
LIN {X 0,Y 752.057,Z 792.984,A -85,B 0,C 180,E1 36024.171,E2 36024.171} C_VEL
LIN {X 0,Y 752.04,Z 815.385,A -85,B 0,C 180,E1 36022.684,E2 36022.684} C_VEL
LIN {X 0,Y 752.063,Z 956.799,A -85,B 0,C 180,E1 36021.311,E2 36021.311} C_VEL
LIN {X 0,Y 752.035,Z 973.627,A -85,B 0,C 180,E1 36020.995,E2 36020.995} C_VEL
LIN {X 0,Y 752.012,Z 989.457,A -85,B 0,C 180,E1 36020.547,E2 36020.547} C_VEL
LIN {X 0,Y 751.992,Z 1005.035,A -85,B 0,C 180,E1 36019.943,E2 36019.943} C_VEL
LIN {X 0,Y 751.987,Z 1018.818,A -85,B 0,C 180,E1 36019.252,E2 36019.252} C_VEL
LIN {X 0,Y 751.966,Z 1032.694,A -85,B 0,C 180,E1 36018.367,E2 36018.367} C_VEL
LIN {X 0,Y 751.945,Z 1044.573,A -85,B 0,C 180,E1 36017.407,E2 36017.407} C_VEL
LIN {X 0,Y 751.926,Z 1054.105,A -85,B 0,C 180,E1 36016.452,E2 36016.452} C_VEL
LIN {X 0,Y 751.925,Z 1062.437,A -85,B 0,C 180,E1 36015.41,E2 36015.41} C_VEL
LIN {X 0,Y 751.92,Z 1070.008,A -85,B 0,C 180,E1 36014.161,E2 36014.161} C_VEL
LIN {X 0,Y 751.916,Z 1075.135,A -85,B 0,C 180,E1 36012.985,E2 36012.985} C_VEL
LIN {X 0,Y 751.915,Z 1078.479,A -85,B 0,C 180,E1 36011.815,E2 36011.815} C_VEL
LIN {X 0,Y 751.916,Z 1080.328,A -85,B 0,C 180,E1 36010.495,E2 36010.495} C_VEL
LIN {X 0,Y 751.918,Z 1080.19,A -85,B 0,C 180,E1 36009.257,E2 36009.257} C_VEL
LIN {X 0,Y 751.915,Z 1078.332,A -85,B 0,C 180,E1 36008.024,E2 36008.024} C_VEL
LIN {X 0,Y 751.916,Z 1074.662,A -85,B 0,C 180,E1 36006.795,E2 36006.795} C_VEL
LIN {X 0,Y 751.921,Z 1068.65,A -85,B 0,C 180,E1 36005.492,E2 36005.492} C_VEL
LIN {X 0,Y 751.924,Z 1061.859,A -85,B 0,C 180,E1 36004.422,E2 36004.422} C_VEL
LIN {X 0,Y 751.927,Z 1053.139,A -85,B 0,C 180,E1 36003.353,E2 36003.353} C_VEL
LIN {X 0,Y 751.949,Z 1043.008,A -85,B 0,C 180,E1 36002.361,E2 36002.361} C_VEL
LIN {X 0,Y 751.968,Z 1029.666,A -85,B 0,C 180,E1 36001.332,E2 36001.332} C_VEL
LIN {X 0,Y 751.99,Z 1017.201,A -85,B 0,C 180,E1 36000.57,E2 36000.57} C_VEL
LIN {X 0,Y 751.963,Z 1003.141,A -85,B 0,C 180,E1 35999.884,E2 35999.884} C_VEL
LIN {X 0,Y 752.014,Z 987.985,A -85,B 0,C 180,E1 35999.313,E2 35999.313} C_VEL
LIN {X 0,Y 752.053,Z 971.91,A -85,B 0,C 180,E1 35998.877,E2 35998.877} C_VEL
LIN {X 0,Y 752.063,Z 955.744,A -85,B 0,C 180,E1 35998.584,E2 35998.584} C_VEL
LIN {X 0,Y 752.023,Z 814.962,A -85,B 0,C 180,E1 35997.217,E2 35997.217} C_VEL
LIN {X 0,Y 752.085,Z 771.926,A -85,B 0,C 180,E1 35994.314,E2 35994.314} C_VEL
LIN {X 0,Y 752.082,Z 732.088,A -85,B 0,C 180,E1 35991.589,E2 35991.589} C_VEL
LIN {X 0,Y 752.176,Z 695.349,A -85,B 0,C 180,E1 35989.04,E2 35989.04} C_VEL
LIN {X 0,Y 752.227,Z 656.378,A -85,B 0,C 180,E1 35986.312,E2 35986.312} C_VEL
LIN {X 0,Y 752.111,Z 624.291,A -85,B 0,C 180,E1 35984.144,E2 35984.144} C_VEL
LIN {X 0,Y 751.941,Z 607.006,A -85,B 0,C 180,E1 35983.012,E2 35983.012} C_VEL
LIN {X 0,Y 751.943,Z 607.004,A -85,B 0,C 180,E1 35980.259,E2 35980.259} C_VEL
LIN {X 0,Y 751.966,Z 607.002,A -85,B 0,C 180,E1 35977.399,E2 35977.399} C_VEL
LIN {X 0,Y 751.958,Z 607.004,A -85,B 0,C 180,E1 35974.534,E2 35974.534} C_VEL
LIN {X 0,Y 751.98,Z 607.003,A -85,B 0,C 180,E1 35971.659,E2 35971.659} C_VEL
LIN {X 0,Y 751.971,Z 607.004,A -85,B 0,C 180,E1 35968.755,E2 35968.755} C_VEL
LIN {X 0,Y 751.974,Z 607.001,A -85,B 0,C 180,E1 35965.865,E2 35965.865} C_VEL
LIN {X 0,Y 751.948,Z 607.004,A -85,B 0,C 180,E1 35963.048,E2 35963.048} C_VEL
LIN {X 0,Y 751.96,Z 607.003,A -85,B 0,C 180,E1 35960.337,E2 35960.337} C_VEL
LIN {X 0,Y 751.974,Z 606.999,A -85,B 0,C 180,E1 35957.404,E2 35957.404} C_VEL
LIN {X 0,Y 751.93,Z 607.004,A -85,B 0,C 180,E1 35954.488,E2 35954.488} C_VEL
LIN {X 0,Y 751.949,Z 607.002,A -85,B 0,C 180,E1 35951.772,E2 35951.772} C_VEL
LIN {X 0,Y 751.956,Z 607,A -85,B 0,C 180,E1 35948.775,E2 35948.775} C_VEL
LIN {X 0,Y 751.926,Z 607.004,A -85,B 0,C 180,E1 35945.996,E2 35945.996} C_VEL
LIN {X 0,Y 751.957,Z 607,A -85,B 0,C 180,E1 35943.217,E2 35943.217} C_VEL
LIN {X 0,Y 751.984,Z 607.083,A -85,B 0,C 180,E1 35941.113,E2 35941.113} C_VEL
LIN {X 0,Y 752.542,Z 610.236,A -85,B 0,C 180,E1 35940.853,E2 35940.853} C_VEL
LIN {X 0,Y 752.423,Z 649.062,A -85,B 0,C 180,E1 35938.017,E2 35938.017} C_VEL
LIN {X 0,Y 752.359,Z 683.189,A -85,B 0,C 180,E1 35935.601,E2 35935.601} C_VEL
LIN {X 0,Y 752.629,Z 691.44,A -85,B 0,C 180,E1 35935.506,E2 35935.506} C_VEL
LIN {X 0,Y 752.498,Z 981.335,A -85,B 0,C 180,E1 35932.531,E2 35932.531} C_VEL
LIN {X 0,Y 752.462,Z 1002.963,A -85,B 0,C 180,E1 35932.204,E2 35932.204} C_VEL
LIN {X 0,Y 752.425,Z 1023.847,A -85,B 0,C 180,E1 35931.751,E2 35931.751} C_VEL
LIN {X 0,Y 752.376,Z 1045.016,A -85,B 0,C 180,E1 35931.15,E2 35931.15} C_VEL
LIN {X 0,Y 752.316,Z 1065.776,A -85,B 0,C 180,E1 35930.418,E2 35930.418} C_VEL
LIN {X 0,Y 752.263,Z 1085.534,A -85,B 0,C 180,E1 35929.568,E2 35929.568} C_VEL
LIN {X 0,Y 752.198,Z 1104.522,A -85,B 0,C 180,E1 35928.596,E2 35928.596} C_VEL
LIN {X 0,Y 752.131,Z 1123.078,A -85,B 0,C 180,E1 35927.483,E2 35927.483} C_VEL
LIN {X 0,Y 752.076,Z 1140.144,A -85,B 0,C 180,E1 35926.29,E2 35926.29} C_VEL
LIN {X 0,Y 752.034,Z 1155.665,A -85,B 0,C 180,E1 35925.025,E2 35925.025} C_VEL
LIN {X 0,Y 751.992,Z 1169.789,A -85,B 0,C 180,E1 35923.689,E2 35923.689} C_VEL
LIN {X 0,Y 751.967,Z 1183.27,A -85,B 0,C 180,E1 35922.204,E2 35922.204} C_VEL
LIN {X 0,Y 751.938,Z 1194.696,A -85,B 0,C 180,E1 35920.728,E2 35920.728} C_VEL
LIN {X 0,Y 751.919,Z 1204.6,A -85,B 0,C 180,E1 35919.181,E2 35919.181} C_VEL
LIN {X 0,Y 751.906,Z 1213.115,A -85,B 0,C 180,E1 35917.564,E2 35917.564} C_VEL
LIN {X 0,Y 751.906,Z 1219.877,A -85,B 0,C 180,E1 35915.953,E2 35915.953} C_VEL
LIN {X 0,Y 751.918,Z 1224.811,A -85,B 0,C 180,E1 35914.346,E2 35914.346} C_VEL
LIN {X 0,Y 751.915,Z 1228.45,A -85,B 0,C 180,E1 35912.59,E2 35912.59} C_VEL
LIN {X 0,Y 751.911,Z 1230.241,A -85,B 0,C 180,E1 35910.913,E2 35910.913} C_VEL
LIN {X 0,Y 751.904,Z 1230.307,A -85,B 0,C 180,E1 35909.313,E2 35909.313} C_VEL
LIN {X 0,Y 751.909,Z 1228.781,A -85,B 0,C 180,E1 35907.636,E2 35907.636} C_VEL
LIN {X 0,Y 751.917,Z 1225.624,A -85,B 0,C 180,E1 35905.958,E2 35905.958} C_VEL
LIN {X 0,Y 751.905,Z 1220.89,A -85,B 0,C 180,E1 35904.352,E2 35904.352} C_VEL
LIN {X 0,Y 751.912,Z 1214.166,A -85,B 0,C 180,E1 35902.665,E2 35902.665} C_VEL
LIN {X 0,Y 751.93,Z 1206.411,A -85,B 0,C 180,E1 35901.123,E2 35901.123} C_VEL
LIN {X 0,Y 751.946,Z 1196.763,A -85,B 0,C 180,E1 35899.58,E2 35899.58} C_VEL
LIN {X 0,Y 751.964,Z 1185.172,A -85,B 0,C 180,E1 35898.027,E2 35898.027} C_VEL
LIN {X 0,Y 751.993,Z 1172.864,A -85,B 0,C 180,E1 35896.622,E2 35896.622} C_VEL
LIN {X 0,Y 752.028,Z 1158.305,A -85,B 0,C 180,E1 35895.209,E2 35895.209} C_VEL
LIN {X 0,Y 752.071,Z 1142.647,A -85,B 0,C 180,E1 35893.906,E2 35893.906} C_VEL
LIN {X 0,Y 752.125,Z 1125.177,A -85,B 0,C 180,E1 35892.656,E2 35892.656} C_VEL
LIN {X 0,Y 752.19,Z 1107.263,A -85,B 0,C 180,E1 35891.555,E2 35891.555} C_VEL
LIN {X 0,Y 752.241,Z 1088.888,A -85,B 0,C 180,E1 35890.591,E2 35890.591} C_VEL
LIN {X 0,Y 752.308,Z 1069.705,A -85,B 0,C 180,E1 35889.742,E2 35889.742} C_VEL
LIN {X 0,Y 752.37,Z 1050.079,A -85,B 0,C 180,E1 35889.012,E2 35889.012} C_VEL
LIN {X 0,Y 752.401,Z 1029.7,A -85,B 0,C 180,E1 35888.4,E2 35888.4} C_VEL
LIN {X 0,Y 752.462,Z 1007.79,A -85,B 0,C 180,E1 35887.892,E2 35887.892} C_VEL
LIN {X 0,Y 752.493,Z 986.505,A -85,B 0,C 180,E1 35887.531,E2 35887.531} C_VEL
LIN {X 0,Y 752.56,Z 876.86,A -85,B 0,C 180,E1 35886.397,E2 35886.397} C_VEL
LIN {X 0,Y 752.512,Z 683.926,A -85,B 0,C 180,E1 35884.412,E2 35884.412} C_VEL
LIN {X 0,Y 752.3,Z 682.479,A -85,B 0,C 180,E1 35884.365,E2 35884.365} C_VEL
LIN {X 0,Y 752.45,Z 646.043,A -85,B 0,C 180,E1 35881.766,E2 35881.766} C_VEL
LIN {X 0,Y 752.553,Z 609.173,A -85,B 0,C 180,E1 35879.068,E2 35879.068} C_VEL
LIN {X 0,Y 751.96,Z 607.001,A -85,B 0,C 180,E1 35878.851,E2 35878.851} C_VEL
LIN {X 0,Y 751.955,Z 607.002,A -85,B 0,C 180,E1 35875.957,E2 35875.957} C_VEL
LIN {X 0,Y 751.971,Z 606.992,A -85,B 0,C 180,E1 35873.05,E2 35873.05} C_VEL
LIN {X 0,Y 751.961,Z 607.003,A -85,B 0,C 180,E1 35869.989,E2 35869.989} C_VEL
LIN {X 0,Y 751.94,Z 606.995,A -85,B 0,C 180,E1 35867.195,E2 35867.195} C_VEL
LIN {X 0,Y 751.97,Z 607,A -85,B 0,C 180,E1 35864.326,E2 35864.326} C_VEL
LIN {X 0,Y 751.926,Z 607,A -85,B 0,C 180,E1 35861.525,E2 35861.525} C_VEL
LIN {X 0,Y 751.94,Z 606.995,A -85,B 0,C 180,E1 35858.877,E2 35858.877} C_VEL
LIN {X 0,Y 751.965,Z 607.004,A -85,B 0,C 180,E1 35855.903,E2 35855.903} C_VEL
LIN {X 0,Y 751.909,Z 607,A -85,B 0,C 180,E1 35853.223,E2 35853.223} C_VEL
LIN {X 0,Y 751.939,Z 606.997,A -85,B 0,C 180,E1 35850.618,E2 35850.618} C_VEL
LIN {X 0,Y 751.927,Z 607.007,A -85,B 0,C 180,E1 35847.567,E2 35847.567} C_VEL
LIN {X 0,Y 751.93,Z 607.214,A -85,B 0,C 180,E1 35847.008,E2 35847.008} C_VEL
LIN {X 0,Y 752.293,Z 612.322,A -85,B 0,C 180,E1 35846.555,E2 35846.555} C_VEL
LIN {X 0,Y 752.312,Z 624.438,A -85,B 0,C 180,E1 35845.545,E2 35845.545} C_VEL
LIN {X 0,Y 752.63,Z 629.238,A -85,B 0,C 180,E1 35845.484,E2 35845.484} C_VEL
LIN {X 0,Y 752.526,Z 890.632,A -85,B 0,C 180,E1 35842.808,E2 35842.808} C_VEL
LIN {X 0,Y 752.496,Z 928.639,A -85,B 0,C 180,E1 35842.394,E2 35842.394} C_VEL
LIN {X 0,Y 752.465,Z 949.784,A -85,B 0,C 180,E1 35842.024,E2 35842.024} C_VEL
LIN {X 0,Y 752.401,Z 971.75,A -85,B 0,C 180,E1 35841.498,E2 35841.498} C_VEL
LIN {X 0,Y 752.342,Z 992.364,A -85,B 0,C 180,E1 35840.867,E2 35840.867} C_VEL
LIN {X 0,Y 752.304,Z 1012.574,A -85,B 0,C 180,E1 35840.096,E2 35840.096} C_VEL
LIN {X 0,Y 752.235,Z 1032.007,A -85,B 0,C 180,E1 35839.208,E2 35839.208} C_VEL
LIN {X 0,Y 752.171,Z 1050.692,A -85,B 0,C 180,E1 35838.205,E2 35838.205} C_VEL
LIN {X 0,Y 752.123,Z 1068.998,A -85,B 0,C 180,E1 35837.047,E2 35837.047} C_VEL
LIN {X 0,Y 752.069,Z 1085.613,A -85,B 0,C 180,E1 35835.817,E2 35835.817} C_VEL
LIN {X 0,Y 752.015,Z 1101.213,A -85,B 0,C 180,E1 35834.477,E2 35834.477} C_VEL
LIN {X 0,Y 751.973,Z 1115.324,A -85,B 0,C 180,E1 35833.066,E2 35833.066} C_VEL
LIN {X 0,Y 751.961,Z 1127.988,A -85,B 0,C 180,E1 35831.584,E2 35831.584} C_VEL
LIN {X 0,Y 751.929,Z 1138.531,A -85,B 0,C 180,E1 35830.111,E2 35830.111} C_VEL
LIN {X 0,Y 751.913,Z 1148.229,A -85,B 0,C 180,E1 35828.49,E2 35828.49} C_VEL
LIN {X 0,Y 751.914,Z 1155.725,A -85,B 0,C 180,E1 35826.952,E2 35826.952} C_VEL
LIN {X 0,Y 751.92,Z 1161.752,A -85,B 0,C 180,E1 35825.343,E2 35825.343} C_VEL
LIN {X 0,Y 751.912,Z 1166.369,A -85,B 0,C 180,E1 35823.661,E2 35823.661} C_VEL
LIN {X 0,Y 751.898,Z 1169.162,A -85,B 0,C 180,E1 35822.059,E2 35822.059} C_VEL
LIN {X 0,Y 751.898,Z 1170.36,A -85,B 0,C 180,E1 35820.459,E2 35820.459} C_VEL
LIN {X 0,Y 751.908,Z 1170.055,A -85,B 0,C 180,E1 35818.783,E2 35818.783} C_VEL
LIN {X 0,Y 751.916,Z 1168.07,A -85,B 0,C 180,E1 35817.105,E2 35817.105} C_VEL
LIN {X 0,Y 751.918,Z 1164.32,A -85,B 0,C 180,E1 35815.425,E2 35815.425} C_VEL
LIN {X 0,Y 751.912,Z 1161.465,A -85,B 0,C 180,E1 35814.48,E2 35814.48} C_VEL
LIN {X 0,Y 750.892,Z 1159.561,A -85,B 0,C 180,E1 35813.912,E2 35813.912} C_VEL
LIN {X 0,Y 744.667,Z 1153.686,A -85,B 0,C 180,E1 35812.418,E2 35812.418} C_VEL
LIN {X 0,Y 743.934,Z 1151.406,A -85,B 0,C 180,E1 35811.938,E2 35811.938} C_VEL
LIN {X 0,Y 743.955,Z 1142.569,A -85,B 0,C 180,E1 35810.33,E2 35810.33} C_VEL
LIN {X 0,Y 743.989,Z 1132.158,A -85,B 0,C 180,E1 35808.765,E2 35808.765} C_VEL
LIN {X 0,Y 744.039,Z 1120.398,A -85,B 0,C 180,E1 35807.27,E2 35807.27} C_VEL
LIN {X 0,Y 744.096,Z 1107.142,A -85,B 0,C 180,E1 35805.846,E2 35805.846} C_VEL
LIN {X 0,Y 744.184,Z 1091.917,A -85,B 0,C 180,E1 35804.444,E2 35804.444} C_VEL
LIN {X 0,Y 744.283,Z 1075.339,A -85,B 0,C 180,E1 35803.133,E2 35803.133} C_VEL
LIN {X 0,Y 744.402,Z 1058.55,A -85,B 0,C 180,E1 35801.989,E2 35801.989} C_VEL
LIN {X 0,Y 744.512,Z 1040.128,A -85,B 0,C 180,E1 35800.914,E2 35800.914} C_VEL
LIN {X 0,Y 744.64,Z 1020.312,A -85,B 0,C 180,E1 35799.938,E2 35799.938} C_VEL
LIN {X 0,Y 744.766,Z 999.438,A -85,B 0,C 180,E1 35799.079,E2 35799.079} C_VEL
LIN {X 0,Y 744.894,Z 978.754,A -85,B 0,C 180,E1 35798.381,E2 35798.381} C_VEL
LIN {X 0,Y 744.984,Z 957.489,A -85,B 0,C 180,E1 35797.822,E2 35797.822} C_VEL
LIN {X 0,Y 745.062,Z 935.074,A -85,B 0,C 180,E1 35797.383,E2 35797.383} C_VEL
LIN {X 0,Y 745.123,Z 913.162,A -85,B 0,C 180,E1 35797.093,E2 35797.093} C_VEL
LIN {X 0,Y 745.445,Z 638.104,A -85,B 0,C 180,E1 35794.255,E2 35794.255} C_VEL
LIN {X 0,Y 745.214,Z 626.379,A -85,B 0,C 180,E1 35794.124,E2 35794.124} C_VEL
LIN {X 0,Y 744.674,Z 623.927,A -85,B 0,C 180,E1 35794.063,E2 35794.063} C_VEL
LIN {X 0,Y 744.627,Z 610.594,A -85,B 0,C 180,E1 35792.909,E2 35792.909} C_VEL
LIN {X 0,Y 744.036,Z 607.991,A -85,B 0,C 180,E1 35792.641,E2 35792.641} C_VEL
LIN {X 0,Y 743.969,Z 607.993,A -85,B 0,C 180,E1 35789.79,E2 35789.79} C_VEL
LIN {X 0,Y 743.947,Z 607.994,A -85,B 0,C 180,E1 35787.39,E2 35787.39} C_VEL
LIN {X 0,Y 744.041,Z 607.989,A -85,B 0,C 180,E1 35784.608,E2 35784.608} C_VEL
LIN {X 0,Y 743.99,Z 607.988,A -85,B 0,C 180,E1 35781.817,E2 35781.817} C_VEL
LIN {X 0,Y 744.026,Z 607.99,A -85,B 0,C 180,E1 35779.049,E2 35779.049} C_VEL
LIN {X 0,Y 744.037,Z 607.982,A -85,B 0,C 180,E1 35776.192,E2 35776.192} C_VEL
LIN {X 0,Y 743.994,Z 607.991,A -85,B 0,C 180,E1 35773.362,E2 35773.362} C_VEL
LIN {X 0,Y 743.957,Z 607.992,A -85,B 0,C 180,E1 35770.832,E2 35770.832} C_VEL
LIN {X 0,Y 744.028,Z 607.99,A -85,B 0,C 180,E1 35767.989,E2 35767.989} C_VEL
LIN {X 0,Y 743.978,Z 607.989,A -85,B 0,C 180,E1 35765.304,E2 35765.304} C_VEL
LIN {X 0,Y 744.035,Z 607.992,A -85,B 0,C 180,E1 35762.588,E2 35762.588} C_VEL
LIN {X 0,Y 744.026,Z 607.984,A -85,B 0,C 180,E1 35759.605,E2 35759.605} C_VEL
LIN {X 0,Y 744.001,Z 607.99,A -85,B 0,C 180,E1 35756.758,E2 35756.758} C_VEL
LIN {X 0,Y 743.982,Z 607.989,A -85,B 0,C 180,E1 35754.116,E2 35754.116} C_VEL
LIN {X 0,Y 743.97,Z 607.993,A -85,B 0,C 180,E1 35751.113,E2 35751.113} C_VEL
LIN {X 0,Y 743.963,Z 607.991,A -85,B 0,C 180,E1 35748.653,E2 35748.653} C_VEL
LIN {X 0,Y 744.035,Z 607.991,A -85,B 0,C 180,E1 35745.912,E2 35745.912} C_VEL
LIN {X 0,Y 744.015,Z 607.984,A -85,B 0,C 180,E1 35743.022,E2 35743.022} C_VEL
LIN {X 0,Y 744.012,Z 607.99,A -85,B 0,C 180,E1 35740.219,E2 35740.219} C_VEL
LIN {X 0,Y 744.012,Z 607.985,A -85,B 0,C 180,E1 35737.414,E2 35737.414} C_VEL
LIN {X 0,Y 743.966,Z 607.993,A -85,B 0,C 180,E1 35734.472,E2 35734.472} C_VEL
LIN {X 0,Y 743.95,Z 607.992,A -85,B 0,C 180,E1 35732.004,E2 35732.004} C_VEL
LIN {X 0,Y 744.038,Z 607.99,A -85,B 0,C 180,E1 35729.308,E2 35729.308} C_VEL
LIN {X 0,Y 744.004,Z 607.985,A -85,B 0,C 180,E1 35726.457,E2 35726.457} C_VEL
LIN {X 0,Y 744.02,Z 607.99,A -85,B 0,C 180,E1 35723.674,E2 35723.674} C_VEL
LIN {X 0,Y 744.032,Z 607.983,A -85,B 0,C 180,E1 35720.799,E2 35720.799} C_VEL
LIN {X 0,Y 743.977,Z 607.991,A -85,B 0,C 180,E1 35717.899,E2 35717.899} C_VEL
LIN {X 0,Y 743.943,Z 607.993,A -85,B 0,C 180,E1 35715.524,E2 35715.524} C_VEL
LIN {X 0,Y 744.035,Z 607.993,A -85,B 0,C 180,E1 35712.832,E2 35712.832} C_VEL
LIN {X 0,Y 743.994,Z 607.987,A -85,B 0,C 180,E1 35709.946,E2 35709.946} C_VEL
LIN {X 0,Y 744.03,Z 607.991,A -85,B 0,C 180,E1 35707.148,E2 35707.148} C_VEL
LIN {X 0,Y 744.037,Z 607.983,A -85,B 0,C 180,E1 35704.19,E2 35704.19} C_VEL
LIN {X 0,Y 743.988,Z 607.991,A -85,B 0,C 180,E1 35701.33,E2 35701.33} C_VEL
LIN {X 0,Y 743.954,Z 607.992,A -85,B 0,C 180,E1 35698.841,E2 35698.841} C_VEL
LIN {X 0,Y 744.029,Z 607.99,A -85,B 0,C 180,E1 35696.009,E2 35696.009} C_VEL
LIN {X 0,Y 743.978,Z 607.989,A -85,B 0,C 180,E1 35693.222,E2 35693.222} C_VEL
LIN {X 0,Y 744.029,Z 607.99,A -85,B 0,C 180,E1 35690.475,E2 35690.475} C_VEL
LIN {X 0,Y 744.024,Z 607.985,A -85,B 0,C 180,E1 35687.54,E2 35687.54} C_VEL
LIN {X 0,Y 743.999,Z 607.991,A -85,B 0,C 180,E1 35684.763,E2 35684.763} C_VEL
LIN {X 0,Y 743.982,Z 607.99,A -85,B 0,C 180,E1 35682.112,E2 35682.112} C_VEL
LIN {X 0,Y 743.959,Z 607.994,A -85,B 0,C 180,E1 35679.031,E2 35679.031} C_VEL
LIN {X 0,Y 743.998,Z 608.04,A -85,B 0,C 180,E1 35677.209,E2 35677.209} C_VEL
LIN {X 0,Y 744.496,Z 612.354,A -85,B 0,C 180,E1 35676.891,E2 35676.891} C_VEL
LIN {X 0,Y 744.572,Z 654.084,A -85,B 0,C 180,E1 35674.006,E2 35674.006} C_VEL
LIN {X 0,Y 744.513,Z 694.027,A -85,B 0,C 180,E1 35671.189,E2 35671.189} C_VEL
LIN {X 0,Y 744.352,Z 734.48,A -85,B 0,C 180,E1 35668.352,E2 35668.352} C_VEL
LIN {X 0,Y 744.225,Z 778.863,A -85,B 0,C 180,E1 35665.289,E2 35665.289} C_VEL
LIN {X 0,Y 744.15,Z 815.397,A -85,B 0,C 180,E1 35662.821,E2 35662.821} C_VEL
LIN {X 0,Y 744.217,Z 956.927,A -85,B 0,C 180,E1 35661.43,E2 35661.43} C_VEL
LIN {X 0,Y 744.172,Z 973.693,A -85,B 0,C 180,E1 35661.111,E2 35661.111} C_VEL
LIN {X 0,Y 744.126,Z 990.191,A -85,B 0,C 180,E1 35660.635,E2 35660.635} C_VEL
LIN {X 0,Y 744.082,Z 1004.579,A -85,B 0,C 180,E1 35660.07,E2 35660.07} C_VEL
LIN {X 0,Y 744.061,Z 1017.48,A -85,B 0,C 180,E1 35659.424,E2 35659.424} C_VEL
LIN {X 0,Y 744.02,Z 1029.95,A -85,B 0,C 180,E1 35658.652,E2 35658.652} C_VEL
LIN {X 0,Y 743.978,Z 1043.342,A -85,B 0,C 180,E1 35657.599,E2 35657.599} C_VEL
LIN {X 0,Y 743.944,Z 1053.281,A -85,B 0,C 180,E1 35656.612,E2 35656.612} C_VEL
LIN {X 0,Y 743.937,Z 1061.526,A -85,B 0,C 180,E1 35655.591,E2 35655.591} C_VEL
LIN {X 0,Y 743.925,Z 1068.603,A -85,B 0,C 180,E1 35654.475,E2 35654.475} C_VEL
LIN {X 0,Y 743.919,Z 1074.44,A -85,B 0,C 180,E1 35653.206,E2 35653.206} C_VEL
LIN {X 0,Y 743.916,Z 1078.056,A -85,B 0,C 180,E1 35652.023,E2 35652.023} C_VEL
LIN {X 0,Y 743.916,Z 1080.032,A -85,B 0,C 180,E1 35650.844,E2 35650.844} C_VEL
LIN {X 0,Y 743.917,Z 1080.381,A -85,B 0,C 180,E1 35649.514,E2 35649.514} C_VEL
LIN {X 0,Y 743.918,Z 1078.866,A -85,B 0,C 180,E1 35648.267,E2 35648.267} C_VEL
LIN {X 0,Y 743.918,Z 1075.574,A -85,B 0,C 180,E1 35647.024,E2 35647.024} C_VEL
LIN {X 0,Y 743.92,Z 1070.79,A -85,B 0,C 180,E1 35645.861,E2 35645.861} C_VEL
LIN {X 0,Y 743.93,Z 1064.176,A -85,B 0,C 180,E1 35644.701,E2 35644.701} C_VEL
LIN {X 0,Y 743.945,Z 1055.473,A -85,B 0,C 180,E1 35643.543,E2 35643.543} C_VEL
LIN {X 0,Y 743.97,Z 1045.841,A -85,B 0,C 180,E1 35642.54,E2 35642.54} C_VEL
LIN {X 0,Y 744.001,Z 1034.834,A -85,B 0,C 180,E1 35641.616,E2 35641.616} C_VEL
LIN {X 0,Y 744.048,Z 1022.389,A -85,B 0,C 180,E1 35640.768,E2 35640.768} C_VEL
LIN {X 0,Y 744.049,Z 1008.048,A -85,B 0,C 180,E1 35639.998,E2 35639.998} C_VEL
LIN {X 0,Y 744.093,Z 994.278,A -85,B 0,C 180,E1 35639.421,E2 35639.421} C_VEL
LIN {X 0,Y 744.179,Z 979.249,A -85,B 0,C 180,E1 35638.94,E2 35638.94} C_VEL
LIN {X 0,Y 744.21,Z 961.628,A -85,B 0,C 180,E1 35638.552,E2 35638.552} C_VEL
LIN {X 0,Y 744.232,Z 943.162,A -85,B 0,C 180,E1 35638.326,E2 35638.326} C_VEL
LIN {X 0,Y 744.138,Z 814.846,A -85,B 0,C 180,E1 35637.072,E2 35637.072} C_VEL
LIN {X 0,Y 744.258,Z 771.82,A -85,B 0,C 180,E1 35634.138,E2 35634.138} C_VEL
LIN {X 0,Y 744.316,Z 732.553,A -85,B 0,C 180,E1 35631.423,E2 35631.423} C_VEL
LIN {X 0,Y 744.493,Z 695.264,A -85,B 0,C 180,E1 35628.808,E2 35628.808} C_VEL
LIN {X 0,Y 744.481,Z 668.97,A -85,B 0,C 180,E1 35626.989,E2 35626.989} C_VEL
LIN {X 0,Y 744.345,Z 632.382,A -85,B 0,C 180,E1 35624.494,E2 35624.494} C_VEL
LIN {X 0,Y 744.073,Z 608.401,A -85,B 0,C 180,E1 35622.924,E2 35622.924} C_VEL
LIN {X 0,Y 744.015,Z 607.995,A -85,B 0,C 180,E1 35622.882,E2 35622.882} C_VEL
LIN {X 0,Y 744.028,Z 607.993,A -85,B 0,C 180,E1 35620.04,E2 35620.04} C_VEL
LIN {X 0,Y 744.038,Z 607.993,A -85,B 0,C 180,E1 35617.145,E2 35617.145} C_VEL
LIN {X 0,Y 744.034,Z 607.991,A -85,B 0,C 180,E1 35614.187,E2 35614.187} C_VEL
LIN {X 0,Y 744.007,Z 607.993,A -85,B 0,C 180,E1 35611.328,E2 35611.328} C_VEL
LIN {X 0,Y 744.013,Z 607.992,A -85,B 0,C 180,E1 35608.57,E2 35608.57} C_VEL
LIN {X 0,Y 744.035,Z 607.988,A -85,B 0,C 180,E1 35605.636,E2 35605.636} C_VEL
LIN {X 0,Y 743.989,Z 607.993,A -85,B 0,C 180,E1 35602.689,E2 35602.689} C_VEL
LIN {X 0,Y 744.005,Z 607.991,A -85,B 0,C 180,E1 35599.997,E2 35599.997} C_VEL
LIN {X 0,Y 744.019,Z 607.989,A -85,B 0,C 180,E1 35596.944,E2 35596.944} C_VEL
LIN {X 0,Y 743.991,Z 607.992,A -85,B 0,C 180,E1 35594.136,E2 35594.136} C_VEL
LIN {X 0,Y 744.027,Z 607.989,A -85,B 0,C 180,E1 35591.286,E2 35591.286} C_VEL
LIN {X 0,Y 744.017,Z 607.991,A -85,B 0,C 180,E1 35588.379,E2 35588.379} C_VEL
LIN {X 0,Y 744.006,Z 607.993,A -85,B 0,C 180,E1 35585.584,E2 35585.584} C_VEL
LIN {X 0,Y 744.038,Z 607.991,A -85,B 0,C 180,E1 35582.698,E2 35582.698} C_VEL
LIN {X 0,Y 744.029,Z 608.146,A -85,B 0,C 180,E1 35581.404,E2 35581.404} C_VEL
LIN {X 0,Y 745.188,Z 612.625,A -85,B 0,C 180,E1 35581.012,E2 35581.012} C_VEL
LIN {X 0,Y 744.965,Z 650.854,A -85,B 0,C 180,E1 35578.192,E2 35578.192} C_VEL
LIN {X 0,Y 744.833,Z 683.269,A -85,B 0,C 180,E1 35575.878,E2 35575.878} C_VEL
LIN {X 0,Y 745.405,Z 687.525,A -85,B 0,C 180,E1 35575.812,E2 35575.812} C_VEL
LIN {X 0,Y 745.123,Z 972.893,A -85,B 0,C 180,E1 35572.865,E2 35572.865} C_VEL
LIN {X 0,Y 745.061,Z 994.782,A -85,B 0,C 180,E1 35572.577,E2 35572.577} C_VEL
LIN {X 0,Y 744.981,Z 1016.643,A -85,B 0,C 180,E1 35572.153,E2 35572.153} C_VEL
LIN {X 0,Y 744.896,Z 1037.13,A -85,B 0,C 180,E1 35571.62,E2 35571.62} C_VEL
LIN {X 0,Y 744.781,Z 1057.059,A -85,B 0,C 180,E1 35570.963,E2 35570.963} C_VEL
LIN {X 0,Y 744.671,Z 1076.614,A -85,B 0,C 180,E1 35570.185,E2 35570.185} C_VEL
LIN {X 0,Y 744.55,Z 1095.358,A -85,B 0,C 180,E1 35569.289,E2 35569.289} C_VEL
LIN {X 0,Y 744.416,Z 1114.122,A -85,B 0,C 180,E1 35568.236,E2 35568.236} C_VEL
LIN {X 0,Y 744.298,Z 1131.94,A -85,B 0,C 180,E1 35567.068,E2 35567.068} C_VEL
LIN {X 0,Y 744.21,Z 1148.234,A -85,B 0,C 180,E1 35565.826,E2 35565.826} C_VEL
LIN {X 0,Y 744.124,Z 1163.421,A -85,B 0,C 180,E1 35564.472,E2 35564.472} C_VEL
LIN {X 0,Y 744.044,Z 1177.164,A -85,B 0,C 180,E1 35563.047,E2 35563.047} C_VEL
LIN {X 0,Y 743.987,Z 1189.522,A -85,B 0,C 180,E1 35561.549,E2 35561.549} C_VEL
LIN {X 0,Y 743.958,Z 1199.884,A -85,B 0,C 180,E1 35560.061,E2 35560.061} C_VEL
LIN {X 0,Y 743.937,Z 1208.885,A -85,B 0,C 180,E1 35558.501,E2 35558.501} C_VEL
LIN {X 0,Y 743.916,Z 1216.254,A -85,B 0,C 180,E1 35556.947,E2 35556.947} C_VEL
LIN {X 0,Y 743.915,Z 1222.162,A -85,B 0,C 180,E1 35555.32,E2 35555.32} C_VEL
LIN {X 0,Y 743.915,Z 1226.625,A -85,B 0,C 180,E1 35553.621,E2 35553.621} C_VEL
LIN {X 0,Y 743.918,Z 1229.415,A -85,B 0,C 180,E1 35551.925,E2 35551.925} C_VEL
LIN {X 0,Y 743.903,Z 1230.44,A -85,B 0,C 180,E1 35550.23,E2 35550.23} C_VEL
LIN {X 0,Y 743.899,Z 1229.814,A -85,B 0,C 180,E1 35548.536,E2 35548.536} C_VEL
LIN {X 0,Y 743.897,Z 1227.724,A -85,B 0,C 180,E1 35546.917,E2 35546.917} C_VEL
LIN {X 0,Y 743.903,Z 1223.986,A -85,B 0,C 180,E1 35545.296,E2 35545.296} C_VEL
LIN {X 0,Y 743.916,Z 1218.364,A -85,B 0,C 180,E1 35543.594,E2 35543.594} C_VEL
LIN {X 0,Y 743.938,Z 1211.308,A -85,B 0,C 180,E1 35541.964,E2 35541.964} C_VEL
LIN {X 0,Y 743.95,Z 1202.744,A -85,B 0,C 180,E1 35540.405,E2 35540.405} C_VEL
LIN {X 0,Y 743.983,Z 1192.382,A -85,B 0,C 180,E1 35538.84,E2 35538.84} C_VEL
LIN {X 0,Y 744.045,Z 1180.517,A -85,B 0,C 180,E1 35537.329,E2 35537.329} C_VEL
LIN {X 0,Y 744.09,Z 1167.444,A -85,B 0,C 180,E1 35535.922,E2 35535.922} C_VEL
LIN {X 0,Y 744.175,Z 1152.859,A -85,B 0,C 180,E1 35534.571,E2 35534.571} C_VEL
LIN {X 0,Y 744.282,Z 1136.876,A -85,B 0,C 180,E1 35533.291,E2 35533.291} C_VEL
LIN {X 0,Y 744.394,Z 1119.933,A -85,B 0,C 180,E1 35532.12,E2 35532.12} C_VEL
LIN {X 0,Y 744.499,Z 1101.451,A -85,B 0,C 180,E1 35531.033,E2 35531.033} C_VEL
LIN {X 0,Y 744.633,Z 1081.679,A -85,B 0,C 180,E1 35530.046,E2 35530.046} C_VEL
LIN {X 0,Y 744.767,Z 1061.477,A -85,B 0,C 180,E1 35529.199,E2 35529.199} C_VEL
LIN {X 0,Y 744.865,Z 1041.153,A -85,B 0,C 180,E1 35528.501,E2 35528.501} C_VEL
LIN {X 0,Y 744.969,Z 1020.009,A -85,B 0,C 180,E1 35527.927,E2 35527.927} C_VEL
LIN {X 0,Y 745.057,Z 998.371,A -85,B 0,C 180,E1 35527.481,E2 35527.481} C_VEL
LIN {X 0,Y 745.108,Z 977.486,A -85,B 0,C 180,E1 35527.187,E2 35527.187} C_VEL
LIN {X 0,Y 745.404,Z 690.581,A -85,B 0,C 180,E1 35524.22,E2 35524.22} C_VEL
LIN {X 0,Y 745.127,Z 684.612,A -85,B 0,C 180,E1 35524.147,E2 35524.147} C_VEL
LIN {X 0,Y 744.76,Z 682.617,A -85,B 0,C 180,E1 35524.096,E2 35524.096} C_VEL
LIN {X 0,Y 745.014,Z 646.641,A -85,B 0,C 180,E1 35521.502,E2 35521.502} C_VEL
LIN {X 0,Y 745.145,Z 611.936,A -85,B 0,C 180,E1 35518.934,E2 35518.934} C_VEL
LIN {X 0,Y 744.019,Z 607.994,A -85,B 0,C 180,E1 35518.571,E2 35518.571} C_VEL
LIN {X 0,Y 744.005,Z 607.989,A -85,B 0,C 180,E1 35515.744,E2 35515.744} C_VEL
LIN {X 0,Y 744.034,Z 607.982,A -85,B 0,C 180,E1 35512.886,E2 35512.886} C_VEL
LIN {X 0,Y 744.016,Z 607.992,A -85,B 0,C 180,E1 35509.929,E2 35509.929} C_VEL
LIN {X 0,Y 744.011,Z 607.983,A -85,B 0,C 180,E1 35507.049,E2 35507.049} C_VEL
LIN {X 0,Y 744.029,Z 607.993,A -85,B 0,C 180,E1 35504.011,E2 35504.011} C_VEL
LIN {X 0,Y 743.984,Z 607.987,A -85,B 0,C 180,E1 35501.292,E2 35501.292} C_VEL
LIN {X 0,Y 744.035,Z 607.983,A -85,B 0,C 180,E1 35498.543,E2 35498.543} C_VEL
LIN {X 0,Y 743.99,Z 607.991,A -85,B 0,C 180,E1 35495.588,E2 35495.588} C_VEL
LIN {X 0,Y 743.976,Z 607.988,A -85,B 0,C 180,E1 35492.979,E2 35492.979} C_VEL
LIN {X 0,Y 744.038,Z 607.989,A -85,B 0,C 180,E1 35490.174,E2 35490.174} C_VEL
LIN {X 0,Y 743.968,Z 607.998,A -85,B 0,C 180,E1 35487.329,E2 35487.329} C_VEL
LIN {X 0,Y 743.992,Z 608.198,A -85,B 0,C 180,E1 35487.235,E2 35487.235} C_VEL
LIN {X 0,Y 744.692,Z 612.174,A -85,B 0,C 180,E1 35486.861,E2 35486.861} C_VEL
LIN {X 0,Y 744.712,Z 624.43,A -85,B 0,C 180,E1 35485.825,E2 35485.825} C_VEL
LIN {X 0,Y 745.408,Z 628.653,A -85,B 0,C 180,E1 35485.755,E2 35485.755} C_VEL
LIN {X 0,Y 745.151,Z 889.07,A -85,B 0,C 180,E1 35483.064,E2 35483.064} C_VEL
LIN {X 0,Y 745.091,Z 928.571,A -85,B 0,C 180,E1 35482.63,E2 35482.63} C_VEL
LIN {X 0,Y 745.025,Z 949.816,A -85,B 0,C 180,E1 35482.256,E2 35482.256} C_VEL
LIN {X 0,Y 744.91,Z 971.242,A -85,B 0,C 180,E1 35481.74,E2 35481.74} C_VEL
LIN {X 0,Y 744.801,Z 992.412,A -85,B 0,C 180,E1 35481.087,E2 35481.087} C_VEL
LIN {X 0,Y 744.7,Z 1012.595,A -85,B 0,C 180,E1 35480.31,E2 35480.31} C_VEL
LIN {X 0,Y 744.564,Z 1032.024,A -85,B 0,C 180,E1 35479.414,E2 35479.414} C_VEL
LIN {X 0,Y 744.436,Z 1051.371,A -85,B 0,C 180,E1 35478.36,E2 35478.36} C_VEL
LIN {X 0,Y 744.331,Z 1069.593,A -85,B 0,C 180,E1 35477.191,E2 35477.191} C_VEL
LIN {X 0,Y 744.223,Z 1086.635,A -85,B 0,C 180,E1 35475.909,E2 35475.909} C_VEL
LIN {X 0,Y 744.123,Z 1102.071,A -85,B 0,C 180,E1 35474.554,E2 35474.554} C_VEL
LIN {X 0,Y 744.042,Z 1116.036,A -85,B 0,C 180,E1 35473.129,E2 35473.129} C_VEL
LIN {X 0,Y 744.004,Z 1128.578,A -85,B 0,C 180,E1 35471.631,E2 35471.631} C_VEL
LIN {X 0,Y 743.955,Z 1139.053,A -85,B 0,C 180,E1 35470.142,E2 35470.142} C_VEL
LIN {X 0,Y 743.926,Z 1148.639,A -85,B 0,C 180,E1 35468.504,E2 35468.504} C_VEL
LIN {X 0,Y 743.919,Z 1156.062,A -85,B 0,C 180,E1 35466.949,E2 35466.949} C_VEL
LIN {X 0,Y 743.922,Z 1162.008,A -85,B 0,C 180,E1 35465.323,E2 35465.323} C_VEL
LIN {X 0,Y 743.916,Z 1166.686,A -85,B 0,C 180,E1 35463.546,E2 35463.546} C_VEL
LIN {X 0,Y 743.909,Z 1169.441,A -85,B 0,C 180,E1 35461.85,E2 35461.85} C_VEL
LIN {X 0,Y 743.9,Z 1170.427,A -85,B 0,C 180,E1 35460.233,E2 35460.233} C_VEL
LIN {X 0,Y 743.902,Z 1169.856,A -85,B 0,C 180,E1 35458.538,E2 35458.538} C_VEL
LIN {X 0,Y 743.916,Z 1167.666,A -85,B 0,C 180,E1 35456.843,E2 35456.843} C_VEL
LIN {X 0,Y 743.913,Z 1163.706,A -85,B 0,C 180,E1 35455.144,E2 35455.144} C_VEL
LIN {X 0,Y 743.917,Z 1157.949,A -85,B 0,C 180,E1 35453.442,E2 35453.442} C_VEL
LIN {X 0,Y 743.934,Z 1151.406,A -85,B 0,C 180,E1 35451.938,E2 35451.938} C_VEL
LIN {X 0,Y 742.955,Z 1148.617,A -85,B 0,C 180,E1 35451.385,E2 35451.385} C_VEL
LIN {X 0,Y 736.732,Z 1140.786,A -85,B 0,C 180,E1 35449.933,E2 35449.933} C_VEL
LIN {X 0,Y 735.996,Z 1137.825,A -85,B 0,C 180,E1 35449.468,E2 35449.468} C_VEL
LIN {X 0,Y 736.063,Z 1126.842,A -85,B 0,C 180,E1 35447.927,E2 35447.927} C_VEL
LIN {X 0,Y 736.153,Z 1114.032,A -85,B 0,C 180,E1 35446.412,E2 35446.412} C_VEL
LIN {X 0,Y 736.258,Z 1099.671,A -85,B 0,C 180,E1 35444.968,E2 35444.968} C_VEL
LIN {X 0,Y 736.394,Z 1083.498,A -85,B 0,C 180,E1 35443.575,E2 35443.575} C_VEL
LIN {X 0,Y 736.566,Z 1066.186,A -85,B 0,C 180,E1 35442.299,E2 35442.299} C_VEL
LIN {X 0,Y 736.765,Z 1048.133,A -85,B 0,C 180,E1 35441.158,E2 35441.158} C_VEL
LIN {X 0,Y 736.944,Z 1028.935,A -85,B 0,C 180,E1 35440.129,E2 35440.129} C_VEL
LIN {X 0,Y 737.124,Z 1008.889,A -85,B 0,C 180,E1 35439.226,E2 35439.226} C_VEL
LIN {X 0,Y 737.32,Z 987.749,A -85,B 0,C 180,E1 35438.44,E2 35438.44} C_VEL
LIN {X 0,Y 737.477,Z 967.188,A -85,B 0,C 180,E1 35437.824,E2 35437.824} C_VEL
LIN {X 0,Y 737.602,Z 945.636,A -85,B 0,C 180,E1 35437.333,E2 35437.333} C_VEL
LIN {X 0,Y 737.716,Z 922.624,A -85,B 0,C 180,E1 35436.963,E2 35436.963} C_VEL
LIN {X 0,Y 738.23,Z 640.726,A -85,B 0,C 180,E1 35434.013,E2 35434.013} C_VEL
LIN {X 0,Y 738.018,Z 628.018,A -85,B 0,C 180,E1 35433.87,E2 35433.87} C_VEL
LIN {X 0,Y 737.084,Z 623.946,A -85,B 0,C 180,E1 35433.778,E2 35433.778} C_VEL
LIN {X 0,Y 737.03,Z 612.751,A -85,B 0,C 180,E1 35432.797,E2 35432.797} C_VEL
LIN {X 0,Y 736.095,Z 608.981,A -85,B 0,C 180,E1 35432.408,E2 35432.408} C_VEL
LIN {X 0,Y 736.027,Z 608.983,A -85,B 0,C 180,E1 35429.738,E2 35429.738} C_VEL
LIN {X 0,Y 736.015,Z 608.983,A -85,B 0,C 180,E1 35427.272,E2 35427.272} C_VEL
LIN {X 0,Y 736.072,Z 608.977,A -85,B 0,C 180,E1 35424.325,E2 35424.325} C_VEL
LIN {X 0,Y 736.054,Z 608.978,A -85,B 0,C 180,E1 35421.613,E2 35421.613} C_VEL
LIN {X 0,Y 736.081,Z 608.975,A -85,B 0,C 180,E1 35418.793,E2 35418.793} C_VEL
LIN {X 0,Y 736.089,Z 608.976,A -85,B 0,C 180,E1 35415.937,E2 35415.937} C_VEL
LIN {X 0,Y 736.041,Z 608.979,A -85,B 0,C 180,E1 35413.159,E2 35413.159} C_VEL
LIN {X 0,Y 736.033,Z 608.98,A -85,B 0,C 180,E1 35410.593,E2 35410.593} C_VEL
LIN {X 0,Y 736.035,Z 608.98,A -85,B 0,C 180,E1 35407.587,E2 35407.587} C_VEL
LIN {X 0,Y 736.044,Z 608.979,A -85,B 0,C 180,E1 35405.005,E2 35405.005} C_VEL
LIN {X 0,Y 736.089,Z 608.974,A -85,B 0,C 180,E1 35402.174,E2 35402.174} C_VEL
LIN {X 0,Y 736.084,Z 608.977,A -85,B 0,C 180,E1 35399.277,E2 35399.277} C_VEL
LIN {X 0,Y 736.051,Z 608.978,A -85,B 0,C 180,E1 35396.548,E2 35396.548} C_VEL
LIN {X 0,Y 736.079,Z 608.977,A -85,B 0,C 180,E1 35393.794,E2 35393.794} C_VEL
LIN {X 0,Y 736.015,Z 608.982,A -85,B 0,C 180,E1 35390.935,E2 35390.935} C_VEL
LIN {X 0,Y 736.031,Z 608.98,A -85,B 0,C 180,E1 35388.454,E2 35388.454} C_VEL
LIN {X 0,Y 736.095,Z 608.974,A -85,B 0,C 180,E1 35385.603,E2 35385.603} C_VEL
LIN {X 0,Y 736.076,Z 608.976,A -85,B 0,C 180,E1 35382.714,E2 35382.714} C_VEL
LIN {X 0,Y 736.061,Z 608.976,A -85,B 0,C 180,E1 35379.935,E2 35379.935} C_VEL
LIN {X 0,Y 736.101,Z 608.975,A -85,B 0,C 180,E1 35377.101,E2 35377.101} C_VEL
LIN {X 0,Y 736.013,Z 608.981,A -85,B 0,C 180,E1 35374.286,E2 35374.286} C_VEL
LIN {X 0,Y 736.024,Z 608.98,A -85,B 0,C 180,E1 35371.792,E2 35371.792} C_VEL
LIN {X 0,Y 736.082,Z 608.974,A -85,B 0,C 180,E1 35368.834,E2 35368.834} C_VEL
LIN {X 0,Y 736.078,Z 608.978,A -85,B 0,C 180,E1 35365.951,E2 35365.951} C_VEL
LIN {X 0,Y 736.085,Z 608.972,A -85,B 0,C 180,E1 35362.979,E2 35362.979} C_VEL
LIN {X 0,Y 736.063,Z 608.979,A -85,B 0,C 180,E1 35359.909,E2 35359.909} C_VEL
LIN {X 0,Y 736.021,Z 608.979,A -85,B 0,C 180,E1 35357.367,E2 35357.367} C_VEL
LIN {X 0,Y 736.096,Z 608.98,A -85,B 0,C 180,E1 35354.561,E2 35354.561} C_VEL
LIN {X 0,Y 736.035,Z 608.978,A -85,B 0,C 180,E1 35351.794,E2 35351.794} C_VEL
LIN {X 0,Y 736.098,Z 608.981,A -85,B 0,C 180,E1 35349.07,E2 35349.07} C_VEL
LIN {X 0,Y 736.085,Z 608.973,A -85,B 0,C 180,E1 35346.085,E2 35346.085} C_VEL
LIN {X 0,Y 736.06,Z 608.979,A -85,B 0,C 180,E1 35343.182,E2 35343.182} C_VEL
LIN {X 0,Y 736.061,Z 608.977,A -85,B 0,C 180,E1 35340.457,E2 35340.457} C_VEL
LIN {X 0,Y 736.018,Z 608.982,A -85,B 0,C 180,E1 35337.456,E2 35337.456} C_VEL
LIN {X 0,Y 736.025,Z 608.981,A -85,B 0,C 180,E1 35334.998,E2 35334.998} C_VEL
LIN {X 0,Y 736.096,Z 608.976,A -85,B 0,C 180,E1 35332.223,E2 35332.223} C_VEL
LIN {X 0,Y 736.072,Z 608.976,A -85,B 0,C 180,E1 35329.307,E2 35329.307} C_VEL
LIN {X 0,Y 736.064,Z 608.978,A -85,B 0,C 180,E1 35326.498,E2 35326.498} C_VEL
LIN {X 0,Y 736.1,Z 608.975,A -85,B 0,C 180,E1 35323.63,E2 35323.63} C_VEL
LIN {X 0,Y 736.016,Z 608.983,A -85,B 0,C 180,E1 35320.799,E2 35320.799} C_VEL
LIN {X 0,Y 736.015,Z 608.983,A -85,B 0,C 180,E1 35318.375,E2 35318.375} C_VEL
LIN {X 0,Y 736.092,Z 609.105,A -85,B 0,C 180,E1 35317.381,E2 35317.381} C_VEL
LIN {X 0,Y 736.837,Z 613.571,A -85,B 0,C 180,E1 35317.047,E2 35317.047} C_VEL
LIN {X 0,Y 736.898,Z 658.986,A -85,B 0,C 180,E1 35313.893,E2 35313.893} C_VEL
LIN {X 0,Y 736.746,Z 699.109,A -85,B 0,C 180,E1 35311.043,E2 35311.043} C_VEL
LIN {X 0,Y 736.596,Z 738.419,A -85,B 0,C 180,E1 35308.275,E2 35308.275} C_VEL
LIN {X 0,Y 736.363,Z 782.067,A -85,B 0,C 180,E1 35305.235,E2 35305.235} C_VEL
LIN {X 0,Y 736.268,Z 815.416,A -85,B 0,C 180,E1 35302.961,E2 35302.961} C_VEL
LIN {X 0,Y 736.374,Z 956.997,A -85,B 0,C 180,E1 35301.554,E2 35301.554} C_VEL
LIN {X 0,Y 736.314,Z 973.612,A -85,B 0,C 180,E1 35301.234,E2 35301.234} C_VEL
LIN {X 0,Y 736.246,Z 989.992,A -85,B 0,C 180,E1 35300.758,E2 35300.758} C_VEL
LIN {X 0,Y 736.175,Z 1004.57,A -85,B 0,C 180,E1 35300.179,E2 35300.179} C_VEL
LIN {X 0,Y 736.134,Z 1017.619,A -85,B 0,C 180,E1 35299.518,E2 35299.518} C_VEL
LIN {X 0,Y 736.075,Z 1030.079,A -85,B 0,C 180,E1 35298.737,E2 35298.737} C_VEL
LIN {X 0,Y 736.017,Z 1042.991,A -85,B 0,C 180,E1 35297.714,E2 35297.714} C_VEL
LIN {X 0,Y 735.965,Z 1052.791,A -85,B 0,C 180,E1 35296.738,E2 35296.738} C_VEL
LIN {X 0,Y 735.945,Z 1060.689,A -85,B 0,C 180,E1 35295.765,E2 35295.765} C_VEL
LIN {X 0,Y 735.931,Z 1067.688,A -85,B 0,C 180,E1 35294.684,E2 35294.684} C_VEL
LIN {X 0,Y 735.923,Z 1073.707,A -85,B 0,C 180,E1 35293.433,E2 35293.433} C_VEL
LIN {X 0,Y 735.916,Z 1077.792,A -85,B 0,C 180,E1 35292.155,E2 35292.155} C_VEL
LIN {X 0,Y 735.915,Z 1079.896,A -85,B 0,C 180,E1 35290.964,E2 35290.964} C_VEL
LIN {X 0,Y 735.916,Z 1080.435,A -85,B 0,C 180,E1 35289.697,E2 35289.697} C_VEL
LIN {X 0,Y 735.916,Z 1079.083,A -85,B 0,C 180,E1 35288.357,E2 35288.357} C_VEL
LIN {X 0,Y 735.92,Z 1075.923,A -85,B 0,C 180,E1 35287.1,E2 35287.1} C_VEL
LIN {X 0,Y 735.92,Z 1071.277,A -85,B 0,C 180,E1 35285.925,E2 35285.925} C_VEL
LIN {X 0,Y 735.933,Z 1065.346,A -85,B 0,C 180,E1 35284.83,E2 35284.83} C_VEL
LIN {X 0,Y 735.958,Z 1057.008,A -85,B 0,C 180,E1 35283.659,E2 35283.659} C_VEL
LIN {X 0,Y 735.993,Z 1047.793,A -85,B 0,C 180,E1 35282.646,E2 35282.646} C_VEL
LIN {X 0,Y 736.036,Z 1038.121,A -85,B 0,C 180,E1 35281.789,E2 35281.789} C_VEL
LIN {X 0,Y 736.084,Z 1027.643,A -85,B 0,C 180,E1 35281.01,E2 35281.01} C_VEL
LIN {X 0,Y 736.139,Z 1015.455,A -85,B 0,C 180,E1 35280.271,E2 35280.271} C_VEL
LIN {X 0,Y 736.173,Z 1000.99,A -85,B 0,C 180,E1 35279.57,E2 35279.57} C_VEL
LIN {X 0,Y 736.271,Z 986.15,A -85,B 0,C 180,E1 35279.026,E2 35279.026} C_VEL
LIN {X 0,Y 736.332,Z 970.83,A -85,B 0,C 180,E1 35278.615,E2 35278.615} C_VEL
LIN {X 0,Y 736.376,Z 955.298,A -85,B 0,C 180,E1 35278.333,E2 35278.333} C_VEL
LIN {X 0,Y 736.267,Z 815.164,A -85,B 0,C 180,E1 35276.947,E2 35276.947} C_VEL
LIN {X 0,Y 736.435,Z 772.278,A -85,B 0,C 180,E1 35273.997,E2 35273.997} C_VEL
LIN {X 0,Y 736.556,Z 733.017,A -85,B 0,C 180,E1 35271.253,E2 35271.253} C_VEL
LIN {X 0,Y 736.76,Z 696.618,A -85,B 0,C 180,E1 35268.689,E2 35268.689} C_VEL
LIN {X 0,Y 736.725,Z 671.792,A -85,B 0,C 180,E1 35266.978,E2 35266.978} C_VEL
LIN {X 0,Y 736.553,Z 634.43,A -85,B 0,C 180,E1 35264.447,E2 35264.447} C_VEL
LIN {X 0,Y 736.351,Z 610.328,A -85,B 0,C 180,E1 35262.861,E2 35262.861} C_VEL
LIN {X 0,Y 736.09,Z 608.983,A -85,B 0,C 180,E1 35262.751,E2 35262.751} C_VEL
LIN {X 0,Y 736.086,Z 608.982,A -85,B 0,C 180,E1 35259.815,E2 35259.815} C_VEL
LIN {X 0,Y 736.08,Z 608.982,A -85,B 0,C 180,E1 35256.968,E2 35256.968} C_VEL
LIN {X 0,Y 736.094,Z 608.978,A -85,B 0,C 180,E1 35254.054,E2 35254.054} C_VEL
LIN {X 0,Y 736.052,Z 608.982,A -85,B 0,C 180,E1 35251.077,E2 35251.077} C_VEL
LIN {X 0,Y 736.063,Z 608.981,A -85,B 0,C 180,E1 35248.374,E2 35248.374} C_VEL
LIN {X 0,Y 736.092,Z 608.976,A -85,B 0,C 180,E1 35245.401,E2 35245.401} C_VEL
LIN {X 0,Y 736.051,Z 608.982,A -85,B 0,C 180,E1 35242.495,E2 35242.495} C_VEL
LIN {X 0,Y 736.072,Z 608.979,A -85,B 0,C 180,E1 35239.713,E2 35239.713} C_VEL
LIN {X 0,Y 736.081,Z 608.979,A -85,B 0,C 180,E1 35236.725,E2 35236.725} C_VEL
LIN {X 0,Y 736.063,Z 608.981,A -85,B 0,C 180,E1 35233.947,E2 35233.947} C_VEL
LIN {X 0,Y 736.1,Z 608.979,A -85,B 0,C 180,E1 35231,E2 35231} C_VEL
LIN {X 0,Y 736.096,Z 608.981,A -85,B 0,C 180,E1 35228.013,E2 35228.013} C_VEL
LIN {X 0,Y 736.099,Z 608.979,A -85,B 0,C 180,E1 35225.005,E2 35225.005} C_VEL
LIN {X 0,Y 736.054,Z 608.983,A -85,B 0,C 180,E1 35222.04,E2 35222.04} C_VEL
LIN {X 0,Y 736.058,Z 609.042,A -85,B 0,C 180,E1 35221.715,E2 35221.715} C_VEL
LIN {X 0,Y 737.831,Z 615.612,A -85,B 0,C 180,E1 35221.129,E2 35221.129} C_VEL
LIN {X 0,Y 737.506,Z 653.243,A -85,B 0,C 180,E1 35218.326,E2 35218.326} C_VEL
LIN {X 0,Y 737.308,Z 683.269,A -85,B 0,C 180,E1 35216.162,E2 35216.162} C_VEL
LIN {X 0,Y 738.199,Z 688.641,A -85,B 0,C 180,E1 35216.071,E2 35216.071} C_VEL
LIN {X 0,Y 737.747,Z 973.911,A -85,B 0,C 180,E1 35213.096,E2 35213.096} C_VEL
LIN {X 0,Y 737.657,Z 995.587,A -85,B 0,C 180,E1 35212.803,E2 35212.803} C_VEL
LIN {X 0,Y 737.526,Z 1018.33,A -85,B 0,C 180,E1 35212.348,E2 35212.348} C_VEL
LIN {X 0,Y 737.395,Z 1039.329,A -85,B 0,C 180,E1 35211.787,E2 35211.787} C_VEL
LIN {X 0,Y 737.219,Z 1059.414,A -85,B 0,C 180,E1 35211.101,E2 35211.101} C_VEL
LIN {X 0,Y 737.015,Z 1080.198,A -85,B 0,C 180,E1 35210.238,E2 35210.238} C_VEL
LIN {X 0,Y 736.846,Z 1099.467,A -85,B 0,C 180,E1 35209.283,E2 35209.283} C_VEL
LIN {X 0,Y 736.657,Z 1118.091,A -85,B 0,C 180,E1 35208.19,E2 35208.19} C_VEL
LIN {X 0,Y 736.476,Z 1135.252,A -85,B 0,C 180,E1 35207.011,E2 35207.011} C_VEL
LIN {X 0,Y 736.318,Z 1151.954,A -85,B 0,C 180,E1 35205.677,E2 35205.677} C_VEL
LIN {X 0,Y 736.209,Z 1166.692,A -85,B 0,C 180,E1 35204.31,E2 35204.31} C_VEL
LIN {X 0,Y 736.113,Z 1179.982,A -85,B 0,C 180,E1 35202.87,E2 35202.87} C_VEL
LIN {X 0,Y 736.03,Z 1191.821,A -85,B 0,C 180,E1 35201.359,E2 35201.359} C_VEL
LIN {X 0,Y 735.975,Z 1202.297,A -85,B 0,C 180,E1 35199.776,E2 35199.776} C_VEL
LIN {X 0,Y 735.954,Z 1210.915,A -85,B 0,C 180,E1 35198.2,E2 35198.2} C_VEL
LIN {X 0,Y 735.912,Z 1217.767,A -85,B 0,C 180,E1 35196.631,E2 35196.631} C_VEL
LIN {X 0,Y 735.902,Z 1223.376,A -85,B 0,C 180,E1 35194.988,E2 35194.988} C_VEL
LIN {X 0,Y 735.903,Z 1227.257,A -85,B 0,C 180,E1 35193.348,E2 35193.348} C_VEL
LIN {X 0,Y 735.907,Z 1229.683,A -85,B 0,C 180,E1 35191.634,E2 35191.634} C_VEL
LIN {X 0,Y 735.912,Z 1230.484,A -85,B 0,C 180,E1 35189.921,E2 35189.921} C_VEL
LIN {X 0,Y 735.916,Z 1229.548,A -85,B 0,C 180,E1 35188.208,E2 35188.208} C_VEL
LIN {X 0,Y 735.911,Z 1226.936,A -85,B 0,C 180,E1 35186.494,E2 35186.494} C_VEL
LIN {X 0,Y 735.91,Z 1222.86,A -85,B 0,C 180,E1 35184.837,E2 35184.837} C_VEL
LIN {X 0,Y 735.913,Z 1217.154,A -85,B 0,C 180,E1 35183.21,E2 35183.21} C_VEL
LIN {X 0,Y 735.95,Z 1209.528,A -85,B 0,C 180,E1 35181.531,E2 35181.531} C_VEL
LIN {X 0,Y 735.983,Z 1200.893,A -85,B 0,C 180,E1 35179.985,E2 35179.985} C_VEL
LIN {X 0,Y 736.029,Z 1190.074,A -85,B 0,C 180,E1 35178.4,E2 35178.4} C_VEL
LIN {X 0,Y 736.112,Z 1177.852,A -85,B 0,C 180,E1 35176.888,E2 35176.888} C_VEL
LIN {X 0,Y 736.23,Z 1164.243,A -85,B 0,C 180,E1 35175.448,E2 35175.448} C_VEL
LIN {X 0,Y 736.367,Z 1148.517,A -85,B 0,C 180,E1 35174.024,E2 35174.024} C_VEL
LIN {X 0,Y 736.511,Z 1131.967,A -85,B 0,C 180,E1 35172.748,E2 35172.748} C_VEL
LIN {X 0,Y 736.678,Z 1114.088,A -85,B 0,C 180,E1 35171.563,E2 35171.563} C_VEL
LIN {X 0,Y 736.885,Z 1094.516,A -85,B 0,C 180,E1 35170.458,E2 35170.458} C_VEL
LIN {X 0,Y 737.09,Z 1075.399,A -85,B 0,C 180,E1 35169.543,E2 35169.543} C_VEL
LIN {X 0,Y 737.237,Z 1055.882,A -85,B 0,C 180,E1 35168.769,E2 35168.769} C_VEL
LIN {X 0,Y 737.416,Z 1033.969,A -85,B 0,C 180,E1 35168.06,E2 35168.06} C_VEL
LIN {X 0,Y 737.588,Z 1012.862,A -85,B 0,C 180,E1 35167.524,E2 35167.524} C_VEL
LIN {X 0,Y 737.667,Z 991.559,A -85,B 0,C 180,E1 35167.132,E2 35167.132} C_VEL
LIN {X 0,Y 737.773,Z 962.746,A -85,B 0,C 180,E1 35166.789,E2 35166.789} C_VEL
LIN {X 0,Y 738.195,Z 687.226,A -85,B 0,C 180,E1 35163.914,E2 35163.914} C_VEL
LIN {X 0,Y 737.237,Z 682.727,A -85,B 0,C 180,E1 35163.82,E2 35163.82} C_VEL
LIN {X 0,Y 737.582,Z 646.64,A -85,B 0,C 180,E1 35161.188,E2 35161.188} C_VEL
LIN {X 0,Y 737.744,Z 614.534,A -85,B 0,C 180,E1 35158.785,E2 35158.785} C_VEL
LIN {X 0,Y 736.098,Z 608.982,A -85,B 0,C 180,E1 35158.264,E2 35158.264} C_VEL
LIN {X 0,Y 736.076,Z 608.973,A -85,B 0,C 180,E1 35155.307,E2 35155.307} C_VEL
LIN {X 0,Y 736.093,Z 608.981,A -85,B 0,C 180,E1 35152.318,E2 35152.318} C_VEL
LIN {X 0,Y 736.057,Z 608.977,A -85,B 0,C 180,E1 35149.508,E2 35149.508} C_VEL
LIN {X 0,Y 736.096,Z 608.972,A -85,B 0,C 180,E1 35146.687,E2 35146.687} C_VEL
LIN {X 0,Y 736.061,Z 608.98,A -85,B 0,C 180,E1 35143.723,E2 35143.723} C_VEL
LIN {X 0,Y 736.063,Z 608.974,A -85,B 0,C 180,E1 35140.949,E2 35140.949} C_VEL
LIN {X 0,Y 736.095,Z 608.982,A -85,B 0,C 180,E1 35137.978,E2 35137.978} C_VEL
LIN {X 0,Y 736.036,Z 608.978,A -85,B 0,C 180,E1 35135.266,E2 35135.266} C_VEL
LIN {X 0,Y 736.079,Z 608.975,A -85,B 0,C 180,E1 35132.544,E2 35132.544} C_VEL
LIN {X 0,Y 736.047,Z 608.984,A -85,B 0,C 180,E1 35129.547,E2 35129.547} C_VEL
LIN {X 0,Y 736.069,Z 609.199,A -85,B 0,C 180,E1 35127.465,E2 35127.465} C_VEL
LIN {X 0,Y 737.114,Z 614.667,A -85,B 0,C 180,E1 35126.942,E2 35126.942} C_VEL
LIN {X 0,Y 737.116,Z 624.358,A -85,B 0,C 180,E1 35126.113,E2 35126.113} C_VEL
LIN {X 0,Y 738.2,Z 629.976,A -85,B 0,C 180,E1 35126.012,E2 35126.012} C_VEL
LIN {X 0,Y 737.789,Z 891.244,A -85,B 0,C 180,E1 35123.285,E2 35123.285} C_VEL
LIN {X 0,Y 737.696,Z 928.835,A -85,B 0,C 180,E1 35122.866,E2 35122.866} C_VEL
LIN {X 0,Y 737.597,Z 950.108,A -85,B 0,C 180,E1 35122.487,E2 35122.487} C_VEL
LIN {X 0,Y 737.427,Z 971.729,A -85,B 0,C 180,E1 35121.959,E2 35121.959} C_VEL
LIN {X 0,Y 737.263,Z 992.922,A -85,B 0,C 180,E1 35121.295,E2 35121.295} C_VEL
LIN {X 0,Y 737.101,Z 1013.61,A -85,B 0,C 180,E1 35120.487,E2 35120.487} C_VEL
LIN {X 0,Y 736.896,Z 1032.844,A -85,B 0,C 180,E1 35119.583,E2 35119.583} C_VEL
LIN {X 0,Y 736.706,Z 1052.046,A -85,B 0,C 180,E1 35118.519,E2 35118.519} C_VEL
LIN {X 0,Y 736.54,Z 1070.162,A -85,B 0,C 180,E1 35117.338,E2 35117.338} C_VEL
LIN {X 0,Y 736.383,Z 1087.152,A -85,B 0,C 180,E1 35116.042,E2 35116.042} C_VEL
LIN {X 0,Y 736.237,Z 1102.079,A -85,B 0,C 180,E1 35114.714,E2 35114.714} C_VEL
LIN {X 0,Y 736.118,Z 1116.043,A -85,B 0,C 180,E1 35113.272,E2 35113.272} C_VEL
LIN {X 0,Y 736.054,Z 1128.58,A -85,B 0,C 180,E1 35111.759,E2 35111.759} C_VEL
LIN {X 0,Y 735.986,Z 1139.058,A -85,B 0,C 180,E1 35110.253,E2 35110.253} C_VEL
LIN {X 0,Y 735.942,Z 1148.643,A -85,B 0,C 180,E1 35108.597,E2 35108.597} C_VEL
LIN {X 0,Y 735.924,Z 1156.371,A -85,B 0,C 180,E1 35106.947,E2 35106.947} C_VEL
LIN {X 0,Y 735.924,Z 1162.264,A -85,B 0,C 180,E1 35105.303,E2 35105.303} C_VEL
LIN {X 0,Y 735.915,Z 1166.688,A -85,B 0,C 180,E1 35103.585,E2 35103.585} C_VEL
LIN {X 0,Y 735.907,Z 1169.44,A -85,B 0,C 180,E1 35101.87,E2 35101.87} C_VEL
LIN {X 0,Y 735.901,Z 1170.427,A -85,B 0,C 180,E1 35100.235,E2 35100.235} C_VEL
LIN {X 0,Y 735.903,Z 1169.856,A -85,B 0,C 180,E1 35098.522,E2 35098.522} C_VEL
LIN {X 0,Y 735.916,Z 1167.667,A -85,B 0,C 180,E1 35096.808,E2 35096.808} C_VEL
LIN {X 0,Y 735.915,Z 1163.706,A -85,B 0,C 180,E1 35095.091,E2 35095.091} C_VEL
LIN {X 0,Y 735.922,Z 1157.948,A -85,B 0,C 180,E1 35093.37,E2 35093.37} C_VEL
LIN {X 0,Y 735.94,Z 1150.751,A -85,B 0,C 180,E1 35091.721,E2 35091.721} C_VEL
LIN {X 0,Y 735.977,Z 1142.107,A -85,B 0,C 180,E1 35090.145,E2 35090.145} C_VEL
LIN {X 0,Y 735.996,Z 1137.825,A -85,B 0,C 180,E1 35089.468,E2 35089.468} C_VEL
LIN {X 0,Y 735.022,Z 1134.393,A -85,B 0,C 180,E1 35088.934,E2 35088.934} C_VEL
LIN {X 0,Y 728.866,Z 1124.672,A -85,B 0,C 180,E1 35087.532,E2 35087.532} C_VEL
LIN {X 0,Y 728.171,Z 1121.198,A -85,B 0,C 180,E1 35087.086,E2 35087.086} C_VEL
LIN {X 0,Y 728.296,Z 1107.914,A -85,B 0,C 180,E1 35085.613,E2 35085.613} C_VEL
LIN {X 0,Y 728.468,Z 1092.497,A -85,B 0,C 180,E1 35084.151,E2 35084.151} C_VEL
LIN {X 0,Y 728.672,Z 1075.887,A -85,B 0,C 180,E1 35082.802,E2 35082.802} C_VEL
LIN {X 0,Y 728.922,Z 1058.181,A -85,B 0,C 180,E1 35081.57,E2 35081.57} C_VEL
LIN {X 0,Y 729.174,Z 1039.344,A -85,B 0,C 180,E1 35080.455,E2 35080.455} C_VEL
LIN {X 0,Y 729.423,Z 1019.414,A -85,B 0,C 180,E1 35079.458,E2 35079.458} C_VEL
LIN {X 0,Y 729.672,Z 998.307,A -85,B 0,C 180,E1 35078.583,E2 35078.583} C_VEL
LIN {X 0,Y 729.932,Z 977.28,A -85,B 0,C 180,E1 35077.873,E2 35077.873} C_VEL
LIN {X 0,Y 730.113,Z 956.057,A -85,B 0,C 180,E1 35077.312,E2 35077.312} C_VEL
LIN {X 0,Y 730.274,Z 934.179,A -85,B 0,C 180,E1 35076.885,E2 35076.885} C_VEL
LIN {X 0,Y 730.395,Z 910.768,A -85,B 0,C 180,E1 35076.579,E2 35076.579} C_VEL
LIN {X 0,Y 731.041,Z 635.965,A -85,B 0,C 180,E1 35073.688,E2 35073.688} C_VEL
LIN {X 0,Y 730.773,Z 629.248,A -85,B 0,C 180,E1 35073.605,E2 35073.605} C_VEL
LIN {X 0,Y 729.504,Z 623.964,A -85,B 0,C 180,E1 35073.486,E2 35073.486} C_VEL
LIN {X 0,Y 729.343,Z 614.735,A -85,B 0,C 180,E1 35072.663,E2 35072.663} C_VEL
LIN {X 0,Y 728.158,Z 609.971,A -85,B 0,C 180,E1 35072.169,E2 35072.169} C_VEL
LIN {X 0,Y 728.083,Z 609.971,A -85,B 0,C 180,E1 35069.463,E2 35069.463} C_VEL
LIN {X 0,Y 728.151,Z 609.971,A -85,B 0,C 180,E1 35066.685,E2 35066.685} C_VEL
LIN {X 0,Y 728.095,Z 609.968,A -85,B 0,C 180,E1 35063.809,E2 35063.809} C_VEL
LIN {X 0,Y 728.158,Z 609.969,A -85,B 0,C 180,E1 35061.033,E2 35061.033} C_VEL
LIN {X 0,Y 728.144,Z 609.962,A -85,B 0,C 180,E1 35058.033,E2 35058.033} C_VEL
LIN {X 0,Y 728.126,Z 609.968,A -85,B 0,C 180,E1 35055.217,E2 35055.217} C_VEL
LIN {X 0,Y 728.12,Z 609.966,A -85,B 0,C 180,E1 35052.491,E2 35052.491} C_VEL
LIN {X 0,Y 728.084,Z 609.971,A -85,B 0,C 180,E1 35049.483,E2 35049.483} C_VEL
LIN {X 0,Y 728.087,Z 609.97,A -85,B 0,C 180,E1 35046.944,E2 35046.944} C_VEL
LIN {X 0,Y 728.158,Z 609.964,A -85,B 0,C 180,E1 35044.108,E2 35044.108} C_VEL
LIN {X 0,Y 728.134,Z 609.966,A -85,B 0,C 180,E1 35041.179,E2 35041.179} C_VEL
LIN {X 0,Y 728.126,Z 609.965,A -85,B 0,C 180,E1 35038.369,E2 35038.369} C_VEL
LIN {X 0,Y 728.16,Z 609.966,A -85,B 0,C 180,E1 35035.456,E2 35035.456} C_VEL
LIN {X 0,Y 728.075,Z 609.97,A -85,B 0,C 180,E1 35032.701,E2 35032.701} C_VEL
LIN {X 0,Y 728.093,Z 609.971,A -85,B 0,C 180,E1 35030.164,E2 35030.164} C_VEL
LIN {X 0,Y 728.117,Z 609.965,A -85,B 0,C 180,E1 35027.091,E2 35027.091} C_VEL
LIN {X 0,Y 728.157,Z 609.97,A -85,B 0,C 180,E1 35024.208,E2 35024.208} C_VEL
LIN {X 0,Y 728.155,Z 609.961,A -85,B 0,C 180,E1 35021.165,E2 35021.165} C_VEL
LIN {X 0,Y 728.12,Z 609.968,A -85,B 0,C 180,E1 35018.291,E2 35018.291} C_VEL
LIN {X 0,Y 728.096,Z 609.968,A -85,B 0,C 180,E1 35015.675,E2 35015.675} C_VEL
LIN {X 0,Y 728.098,Z 609.969,A -85,B 0,C 180,E1 35012.677,E2 35012.677} C_VEL
LIN {X 0,Y 728.094,Z 609.968,A -85,B 0,C 180,E1 35010.08,E2 35010.08} C_VEL
LIN {X 0,Y 728.154,Z 609.965,A -85,B 0,C 180,E1 35007.325,E2 35007.325} C_VEL
LIN {X 0,Y 728.138,Z 609.963,A -85,B 0,C 180,E1 35004.406,E2 35004.406} C_VEL
LIN {X 0,Y 728.124,Z 609.967,A -85,B 0,C 180,E1 35001.631,E2 35001.631} C_VEL
LIN {X 0,Y 728.141,Z 609.962,A -85,B 0,C 180,E1 34998.837,E2 34998.837} C_VEL
LIN {X 0,Y 728.08,Z 609.971,A -85,B 0,C 180,E1 34995.933,E2 34995.933} C_VEL
LIN {X 0,Y 728.08,Z 609.97,A -85,B 0,C 180,E1 34993.486,E2 34993.486} C_VEL
LIN {X 0,Y 728.159,Z 609.965,A -85,B 0,C 180,E1 34990.676,E2 34990.676} C_VEL
LIN {X 0,Y 728.129,Z 609.965,A -85,B 0,C 180,E1 34987.814,E2 34987.814} C_VEL
LIN {X 0,Y 728.131,Z 609.966,A -85,B 0,C 180,E1 34984.98,E2 34984.98} C_VEL
LIN {X 0,Y 728.16,Z 609.964,A -85,B 0,C 180,E1 34982.081,E2 34982.081} C_VEL
LIN {X 0,Y 728.084,Z 609.97,A -85,B 0,C 180,E1 34979.277,E2 34979.277} C_VEL
LIN {X 0,Y 728.081,Z 609.971,A -85,B 0,C 180,E1 34976.775,E2 34976.775} C_VEL
LIN {X 0,Y 728.136,Z 609.964,A -85,B 0,C 180,E1 34973.811,E2 34973.811} C_VEL
LIN {X 0,Y 728.128,Z 609.968,A -85,B 0,C 180,E1 34971.005,E2 34971.005} C_VEL
LIN {X 0,Y 728.144,Z 609.962,A -85,B 0,C 180,E1 34968.093,E2 34968.093} C_VEL
LIN {X 0,Y 728.156,Z 609.97,A -85,B 0,C 180,E1 34965.107,E2 34965.107} C_VEL
LIN {X 0,Y 728.091,Z 609.969,A -85,B 0,C 180,E1 34962.37,E2 34962.37} C_VEL
LIN {X 0,Y 728.152,Z 609.971,A -85,B 0,C 180,E1 34959.577,E2 34959.577} C_VEL
LIN {X 0,Y 728.184,Z 610.16,A -85,B 0,C 180,E1 34957.562,E2 34957.562} C_VEL
LIN {X 0,Y 729.176,Z 615.457,A -85,B 0,C 180,E1 34957.157,E2 34957.157} C_VEL
LIN {X 0,Y 729.186,Z 661.395,A -85,B 0,C 180,E1 34953.946,E2 34953.946} C_VEL
LIN {X 0,Y 728.99,Z 700.745,A -85,B 0,C 180,E1 34951.135,E2 34951.135} C_VEL
LIN {X 0,Y 728.827,Z 741.417,A -85,B 0,C 180,E1 34948.269,E2 34948.269} C_VEL
LIN {X 0,Y 728.512,Z 784.253,A -85,B 0,C 180,E1 34945.251,E2 34945.251} C_VEL
LIN {X 0,Y 728.387,Z 815.39,A -85,B 0,C 180,E1 34943.104,E2 34943.104} C_VEL
LIN {X 0,Y 728.685,Z 827.791,A -85,B 0,C 180,E1 34942.976,E2 34942.976} C_VEL
LIN {X 0,Y 728.534,Z 956.984,A -85,B 0,C 180,E1 34941.68,E2 34941.68} C_VEL
LIN {X 0,Y 728.459,Z 973.517,A -85,B 0,C 180,E1 34941.359,E2 34941.359} C_VEL
LIN {X 0,Y 728.369,Z 990.26,A -85,B 0,C 180,E1 34940.867,E2 34940.867} C_VEL
LIN {X 0,Y 728.27,Z 1004.74,A -85,B 0,C 180,E1 34940.282,E2 34940.282} C_VEL
LIN {X 0,Y 728.212,Z 1017.017,A -85,B 0,C 180,E1 34939.656,E2 34939.656} C_VEL
LIN {X 0,Y 728.139,Z 1028.351,A -85,B 0,C 180,E1 34938.949,E2 34938.949} C_VEL
LIN {X 0,Y 728.076,Z 1039.03,A -85,B 0,C 180,E1 34938.138,E2 34938.138} C_VEL
LIN {X 0,Y 728.009,Z 1050.386,A -85,B 0,C 180,E1 34937.081,E2 34937.081} C_VEL
LIN {X 0,Y 727.962,Z 1059.257,A -85,B 0,C 180,E1 34936.024,E2 34936.024} C_VEL
LIN {X 0,Y 727.938,Z 1065.866,A -85,B 0,C 180,E1 34935.045,E2 34935.045} C_VEL
LIN {X 0,Y 727.924,Z 1071.455,A -85,B 0,C 180,E1 34933.988,E2 34933.988} C_VEL
LIN {X 0,Y 727.918,Z 1075.875,A -85,B 0,C 180,E1 34932.856,E2 34932.856} C_VEL
LIN {X 0,Y 727.918,Z 1079.093,A -85,B 0,C 180,E1 34931.567,E2 34931.567} C_VEL
LIN {X 0,Y 727.915,Z 1080.434,A -85,B 0,C 180,E1 34930.205,E2 34930.205} C_VEL
LIN {X 0,Y 727.916,Z 1079.96,A -85,B 0,C 180,E1 34929.007,E2 34929.007} C_VEL
LIN {X 0,Y 727.917,Z 1077.969,A -85,B 0,C 180,E1 34927.814,E2 34927.814} C_VEL
LIN {X 0,Y 727.923,Z 1074.415,A -85,B 0,C 180,E1 34926.624,E2 34926.624} C_VEL
LIN {X 0,Y 727.934,Z 1068.278,A -85,B 0,C 180,E1 34925.279,E2 34925.279} C_VEL
LIN {X 0,Y 727.956,Z 1061.345,A -85,B 0,C 180,E1 34924.173,E2 34924.173} C_VEL
LIN {X 0,Y 727.98,Z 1053.912,A -85,B 0,C 180,E1 34923.226,E2 34923.226} C_VEL
LIN {X 0,Y 728.035,Z 1044.801,A -85,B 0,C 180,E1 34922.281,E2 34922.281} C_VEL
LIN {X 0,Y 728.117,Z 1032.594,A -85,B 0,C 180,E1 34921.257,E2 34921.257} C_VEL
LIN {X 0,Y 728.2,Z 1019.443,A -85,B 0,C 180,E1 34920.392,E2 34920.392} C_VEL
LIN {X 0,Y 728.23,Z 1007.616,A -85,B 0,C 180,E1 34919.762,E2 34919.762} C_VEL
LIN {X 0,Y 728.317,Z 994.774,A -85,B 0,C 180,E1 34919.212,E2 34919.212} C_VEL
LIN {X 0,Y 728.425,Z 981.913,A -85,B 0,C 180,E1 34918.779,E2 34918.779} C_VEL
LIN {X 0,Y 728.494,Z 967.493,A -85,B 0,C 180,E1 34918.418,E2 34918.418} C_VEL
LIN {X 0,Y 728.551,Z 951.704,A -85,B 0,C 180,E1 34918.161,E2 34918.161} C_VEL
LIN {X 0,Y 728.468,Z 815.859,A -85,B 0,C 180,E1 34916.812,E2 34916.812} C_VEL
LIN {X 0,Y 728.383,Z 814.615,A -85,B 0,C 180,E1 34916.772,E2 34916.772} C_VEL
LIN {X 0,Y 728.623,Z 771.609,A -85,B 0,C 180,E1 34913.775,E2 34913.775} C_VEL
LIN {X 0,Y 728.819,Z 732.766,A -85,B 0,C 180,E1 34911.025,E2 34911.025} C_VEL
LIN {X 0,Y 729.05,Z 695.656,A -85,B 0,C 180,E1 34908.408,E2 34908.408} C_VEL
LIN {X 0,Y 728.877,Z 654.218,A -85,B 0,C 180,E1 34905.574,E2 34905.574} C_VEL
LIN {X 0,Y 728.713,Z 612.656,A -85,B 0,C 180,E1 34902.818,E2 34902.818} C_VEL
LIN {X 0,Y 728.157,Z 609.971,A -85,B 0,C 180,E1 34902.616,E2 34902.616} C_VEL
LIN {X 0,Y 728.132,Z 609.971,A -85,B 0,C 180,E1 34899.669,E2 34899.669} C_VEL
LIN {X 0,Y 728.133,Z 609.971,A -85,B 0,C 180,E1 34896.873,E2 34896.873} C_VEL
LIN {X 0,Y 728.158,Z 609.966,A -85,B 0,C 180,E1 34893.899,E2 34893.899} C_VEL
LIN {X 0,Y 728.111,Z 609.971,A -85,B 0,C 180,E1 34890.852,E2 34890.852} C_VEL
LIN {X 0,Y 728.122,Z 609.969,A -85,B 0,C 180,E1 34888.174,E2 34888.174} C_VEL
LIN {X 0,Y 728.145,Z 609.967,A -85,B 0,C 180,E1 34885.161,E2 34885.161} C_VEL
LIN {X 0,Y 728.123,Z 609.971,A -85,B 0,C 180,E1 34882.275,E2 34882.275} C_VEL
LIN {X 0,Y 728.157,Z 609.968,A -85,B 0,C 180,E1 34879.39,E2 34879.39} C_VEL
LIN {X 0,Y 728.155,Z 609.97,A -85,B 0,C 180,E1 34876.421,E2 34876.421} C_VEL
LIN {X 0,Y 728.16,Z 609.968,A -85,B 0,C 180,E1 34873.466,E2 34873.466} C_VEL
LIN {X 0,Y 728.125,Z 609.971,A -85,B 0,C 180,E1 34870.505,E2 34870.505} C_VEL
LIN {X 0,Y 728.139,Z 609.968,A -85,B 0,C 180,E1 34867.723,E2 34867.723} C_VEL
LIN {X 0,Y 728.143,Z 609.968,A -85,B 0,C 180,E1 34864.74,E2 34864.74} C_VEL
LIN {X 0,Y 728.121,Z 610.026,A -85,B 0,C 180,E1 34862.025,E2 34862.025} C_VEL
LIN {X 0,Y 730.487,Z 618.001,A -85,B 0,C 180,E1 34861.294,E2 34861.294} C_VEL
LIN {X 0,Y 730.051,Z 655.632,A -85,B 0,C 180,E1 34858.464,E2 34858.464} C_VEL
LIN {X 0,Y 729.806,Z 683.29,A -85,B 0,C 180,E1 34856.452,E2 34856.452} C_VEL
LIN {X 0,Y 731.006,Z 689.87,A -85,B 0,C 180,E1 34856.334,E2 34856.334} C_VEL
LIN {X 0,Y 730.385,Z 974.79,A -85,B 0,C 180,E1 34853.334,E2 34853.334} C_VEL
LIN {X 0,Y 730.264,Z 996.398,A -85,B 0,C 180,E1 34853.034,E2 34853.034} C_VEL
LIN {X 0,Y 730.085,Z 1019.021,A -85,B 0,C 180,E1 34852.571,E2 34852.571} C_VEL
LIN {X 0,Y 729.904,Z 1039.746,A -85,B 0,C 180,E1 34852.008,E2 34852.008} C_VEL
LIN {X 0,Y 729.673,Z 1059.704,A -85,B 0,C 180,E1 34851.319,E2 34851.319} C_VEL
LIN {X 0,Y 729.406,Z 1080.201,A -85,B 0,C 180,E1 34850.459,E2 34850.459} C_VEL
LIN {X 0,Y 729.179,Z 1099.283,A -85,B 0,C 180,E1 34849.504,E2 34849.504} C_VEL
LIN {X 0,Y 728.928,Z 1117.104,A -85,B 0,C 180,E1 34848.451,E2 34848.451} C_VEL
LIN {X 0,Y 728.681,Z 1134.701,A -85,B 0,C 180,E1 34847.24,E2 34847.24} C_VEL
LIN {X 0,Y 728.481,Z 1151.026,A -85,B 0,C 180,E1 34845.932,E2 34845.932} C_VEL
LIN {X 0,Y 728.329,Z 1165.918,A -85,B 0,C 180,E1 34844.549,E2 34844.549} C_VEL
LIN {X 0,Y 728.18,Z 1179.28,A -85,B 0,C 180,E1 34843.094,E2 34843.094} C_VEL
LIN {X 0,Y 728.069,Z 1191.245,A -85,B 0,C 180,E1 34841.565,E2 34841.565} C_VEL
LIN {X 0,Y 728.001,Z 1201.837,A -85,B 0,C 180,E1 34839.964,E2 34839.964} C_VEL
LIN {X 0,Y 727.966,Z 1210.509,A -85,B 0,C 180,E1 34838.371,E2 34838.371} C_VEL
LIN {X 0,Y 727.917,Z 1217.767,A -85,B 0,C 180,E1 34836.704,E2 34836.704} C_VEL
LIN {X 0,Y 727.905,Z 1223.375,A -85,B 0,C 180,E1 34835.042,E2 34835.042} C_VEL
LIN {X 0,Y 727.905,Z 1227.257,A -85,B 0,C 180,E1 34833.385,E2 34833.385} C_VEL
LIN {X 0,Y 727.908,Z 1229.683,A -85,B 0,C 180,E1 34831.652,E2 34831.652} C_VEL
LIN {X 0,Y 727.913,Z 1230.484,A -85,B 0,C 180,E1 34829.92,E2 34829.92} C_VEL
LIN {X 0,Y 727.917,Z 1229.548,A -85,B 0,C 180,E1 34828.188,E2 34828.188} C_VEL
LIN {X 0,Y 727.913,Z 1226.937,A -85,B 0,C 180,E1 34826.455,E2 34826.455} C_VEL
LIN {X 0,Y 727.914,Z 1222.914,A -85,B 0,C 180,E1 34824.797,E2 34824.797} C_VEL
LIN {X 0,Y 727.917,Z 1217.457,A -85,B 0,C 180,E1 34823.215,E2 34823.215} C_VEL
LIN {X 0,Y 727.961,Z 1209.686,A -85,B 0,C 180,E1 34821.468,E2 34821.468} C_VEL
LIN {X 0,Y 728.01,Z 1200.893,A -85,B 0,C 180,E1 34819.874,E2 34819.874} C_VEL
LIN {X 0,Y 728.075,Z 1190.075,A -85,B 0,C 180,E1 34818.272,E2 34818.272} C_VEL
LIN {X 0,Y 728.184,Z 1177.853,A -85,B 0,C 180,E1 34816.743,E2 34816.743} C_VEL
LIN {X 0,Y 728.345,Z 1164.242,A -85,B 0,C 180,E1 34815.286,E2 34815.286} C_VEL
LIN {X 0,Y 728.522,Z 1149.049,A -85,B 0,C 180,E1 34813.894,E2 34813.894} C_VEL
LIN {X 0,Y 728.723,Z 1132.461,A -85,B 0,C 180,E1 34812.594,E2 34812.594} C_VEL
LIN {X 0,Y 728.942,Z 1114.969,A -85,B 0,C 180,E1 34811.415,E2 34811.415} C_VEL
LIN {X 0,Y 729.214,Z 1096.124,A -85,B 0,C 180,E1 34810.328,E2 34810.328} C_VEL
LIN {X 0,Y 729.478,Z 1076.558,A -85,B 0,C 180,E1 34809.373,E2 34809.373} C_VEL
LIN {X 0,Y 729.692,Z 1057.005,A -85,B 0,C 180,E1 34808.58,E2 34808.58} C_VEL
LIN {X 0,Y 729.935,Z 1035.589,A -85,B 0,C 180,E1 34807.87,E2 34807.87} C_VEL
LIN {X 0,Y 730.152,Z 1014.303,A -85,B 0,C 180,E1 34807.315,E2 34807.315} C_VEL
LIN {X 0,Y 730.277,Z 992.868,A -85,B 0,C 180,E1 34806.909,E2 34806.909} C_VEL
LIN {X 0,Y 730.412,Z 964.909,A -85,B 0,C 180,E1 34806.564,E2 34806.564} C_VEL
LIN {X 0,Y 730.997,Z 688.656,A -85,B 0,C 180,E1 34803.652,E2 34803.652} C_VEL
LIN {X 0,Y 729.731,Z 682.778,A -85,B 0,C 180,E1 34803.533,E2 34803.533} C_VEL
LIN {X 0,Y 730.168,Z 646.937,A -85,B 0,C 180,E1 34800.89,E2 34800.89} C_VEL
LIN {X 0,Y 730.406,Z 617.371,A -85,B 0,C 180,E1 34798.654,E2 34798.654} C_VEL
LIN {X 0,Y 728.138,Z 609.972,A -85,B 0,C 180,E1 34797.943,E2 34797.943} C_VEL
LIN {X 0,Y 728.157,Z 609.961,A -85,B 0,C 180,E1 34794.971,E2 34794.971} C_VEL
LIN {X 0,Y 728.138,Z 609.97,A -85,B 0,C 180,E1 34791.933,E2 34791.933} C_VEL
LIN {X 0,Y 728.141,Z 609.961,A -85,B 0,C 180,E1 34789.05,E2 34789.05} C_VEL
LIN {X 0,Y 728.148,Z 609.971,A -85,B 0,C 180,E1 34785.985,E2 34785.985} C_VEL
LIN {X 0,Y 728.115,Z 609.964,A -85,B 0,C 180,E1 34783.149,E2 34783.149} C_VEL
LIN {X 0,Y 728.158,Z 609.968,A -85,B 0,C 180,E1 34780.227,E2 34780.227} C_VEL
LIN {X 0,Y 728.105,Z 609.968,A -85,B 0,C 180,E1 34777.462,E2 34777.462} C_VEL
LIN {X 0,Y 728.118,Z 609.965,A -85,B 0,C 180,E1 34774.794,E2 34774.794} C_VEL
LIN {X 0,Y 728.128,Z 609.972,A -85,B 0,C 180,E1 34771.733,E2 34771.733} C_VEL
LIN {X 0,Y 728.086,Z 609.971,A -85,B 0,C 180,E1 34769.089,E2 34769.089} C_VEL
LIN {X 0,Y 728.159,Z 610.201,A -85,B 0,C 180,E1 34767.7,E2 34767.7} C_VEL
LIN {X 0,Y 729.537,Z 616.662,A -85,B 0,C 180,E1 34767.068,E2 34767.068} C_VEL
LIN {X 0,Y 729.566,Z 624.454,A -85,B 0,C 180,E1 34766.403,E2 34766.403} C_VEL
LIN {X 0,Y 731.006,Z 631.427,A -85,B 0,C 180,E1 34766.272,E2 34766.272} C_VEL
LIN {X 0,Y 730.436,Z 893.386,A -85,B 0,C 180,E1 34763.512,E2 34763.512} C_VEL
LIN {X 0,Y 730.314,Z 929.104,A -85,B 0,C 180,E1 34763.107,E2 34763.107} C_VEL
LIN {X 0,Y 730.181,Z 950.53,A -85,B 0,C 180,E1 34762.72,E2 34762.72} C_VEL
LIN {X 0,Y 729.955,Z 972.219,A -85,B 0,C 180,E1 34762.183,E2 34762.183} C_VEL
LIN {X 0,Y 729.736,Z 993.428,A -85,B 0,C 180,E1 34761.507,E2 34761.507} C_VEL
LIN {X 0,Y 729.517,Z 1013.631,A -85,B 0,C 180,E1 34760.71,E2 34760.71} C_VEL
LIN {X 0,Y 729.243,Z 1032.861,A -85,B 0,C 180,E1 34759.797,E2 34759.797} C_VEL
LIN {X 0,Y 728.997,Z 1052.058,A -85,B 0,C 180,E1 34758.722,E2 34758.722} C_VEL
LIN {X 0,Y 728.754,Z 1070.73,A -85,B 0,C 180,E1 34757.488,E2 34757.488} C_VEL
LIN {X 0,Y 728.545,Z 1087.661,A -85,B 0,C 180,E1 34756.178,E2 34756.178} C_VEL
LIN {X 0,Y 728.348,Z 1102.937,A -85,B 0,C 180,E1 34754.795,E2 34754.795} C_VEL
LIN {X 0,Y 728.192,Z 1116.756,A -85,B 0,C 180,E1 34753.339,E2 34753.339} C_VEL
LIN {X 0,Y 728.098,Z 1129.166,A -85,B 0,C 180,E1 34751.809,E2 34751.809} C_VEL
LIN {X 0,Y 728.014,Z 1139.581,A -85,B 0,C 180,E1 34750.287,E2 34750.287} C_VEL
LIN {X 0,Y 727.959,Z 1148.647,A -85,B 0,C 180,E1 34748.692,E2 34748.692} C_VEL
LIN {X 0,Y 727.935,Z 1156.371,A -85,B 0,C 180,E1 34747.024,E2 34747.024} C_VEL
LIN {X 0,Y 727.925,Z 1162.267,A -85,B 0,C 180,E1 34745.361,E2 34745.361} C_VEL
LIN {X 0,Y 727.914,Z 1166.69,A -85,B 0,C 180,E1 34743.624,E2 34743.624} C_VEL
LIN {X 0,Y 727.906,Z 1169.439,A -85,B 0,C 180,E1 34741.891,E2 34741.891} C_VEL
LIN {X 0,Y 727.901,Z 1170.427,A -85,B 0,C 180,E1 34740.238,E2 34740.238} C_VEL
LIN {X 0,Y 727.903,Z 1169.856,A -85,B 0,C 180,E1 34738.506,E2 34738.506} C_VEL
LIN {X 0,Y 727.916,Z 1167.667,A -85,B 0,C 180,E1 34736.773,E2 34736.773} C_VEL
LIN {X 0,Y 727.917,Z 1163.704,A -85,B 0,C 180,E1 34735.037,E2 34735.037} C_VEL
LIN {X 0,Y 727.929,Z 1157.948,A -85,B 0,C 180,E1 34733.297,E2 34733.297} C_VEL
LIN {X 0,Y 727.95,Z 1150.75,A -85,B 0,C 180,E1 34731.63,E2 34731.63} C_VEL
LIN {X 0,Y 727.999,Z 1142.104,A -85,B 0,C 180,E1 34730.036,E2 34730.036} C_VEL
LIN {X 0,Y 728.074,Z 1131.578,A -85,B 0,C 180,E1 34728.435,E2 34728.435} C_VEL
LIN {X 0,Y 728.171,Z 1121.198,A -85,B 0,C 180,E1 34727.086,E2 34727.086} C_VEL
LIN {X 0,Y 727.249,Z 1117.073,A -85,B 0,C 180,E1 34726.573,E2 34726.573} C_VEL
LIN {X 0,Y 721.183,Z 1105.703,A -85,B 0,C 180,E1 34725.236,E2 34725.236} C_VEL
LIN {X 0,Y 720.489,Z 1101.611,A -85,B 0,C 180,E1 34724.82,E2 34724.82} C_VEL
LIN {X 0,Y 720.718,Z 1086.672,A -85,B 0,C 180,E1 34723.468,E2 34723.468} C_VEL
LIN {X 0,Y 720.997,Z 1069.735,A -85,B 0,C 180,E1 34722.155,E2 34722.155} C_VEL
LIN {X 0,Y 721.305,Z 1051.605,A -85,B 0,C 180,E1 34720.953,E2 34720.953} C_VEL
LIN {X 0,Y 721.619,Z 1032.239,A -85,B 0,C 180,E1 34719.861,E2 34719.861} C_VEL
LIN {X 0,Y 721.957,Z 1011.864,A -85,B 0,C 180,E1 34718.896,E2 34718.896} C_VEL
LIN {X 0,Y 722.275,Z 991.467,A -85,B 0,C 180,E1 34718.096,E2 34718.096} C_VEL
LIN {X 0,Y 722.521,Z 970.631,A -85,B 0,C 180,E1 34717.44,E2 34717.44} C_VEL
LIN {X 0,Y 722.784,Z 947.963,A -85,B 0,C 180,E1 34716.891,E2 34716.891} C_VEL
LIN {X 0,Y 722.976,Z 926.342,A -85,B 0,C 180,E1 34716.513,E2 34716.513} C_VEL
LIN {X 0,Y 723.515,Z 744.36,A -85,B 0,C 180,E1 34714.566,E2 34714.566} C_VEL
LIN {X 0,Y 723.695,Z 631.247,A -85,B 0,C 180,E1 34713.349,E2 34713.349} C_VEL
LIN {X 0,Y 721.921,Z 623.932,A -85,B 0,C 180,E1 34713.183,E2 34713.183} C_VEL
LIN {X 0,Y 721.876,Z 617.517,A -85,B 0,C 180,E1 34712.607,E2 34712.607} C_VEL
LIN {X 0,Y 720.191,Z 610.961,A -85,B 0,C 180,E1 34711.926,E2 34711.926} C_VEL
LIN {X 0,Y 720.149,Z 610.961,A -85,B 0,C 180,E1 34709.255,E2 34709.255} C_VEL
LIN {X 0,Y 720.186,Z 610.96,A -85,B 0,C 180,E1 34706.364,E2 34706.364} C_VEL
LIN {X 0,Y 720.157,Z 610.958,A -85,B 0,C 180,E1 34703.639,E2 34703.639} C_VEL
LIN {X 0,Y 720.214,Z 610.955,A -85,B 0,C 180,E1 34700.829,E2 34700.829} C_VEL
LIN {X 0,Y 720.203,Z 610.953,A -85,B 0,C 180,E1 34697.892,E2 34697.892} C_VEL
LIN {X 0,Y 720.181,Z 610.956,A -85,B 0,C 180,E1 34695.079,E2 34695.079} C_VEL
LIN {X 0,Y 720.211,Z 610.954,A -85,B 0,C 180,E1 34692.218,E2 34692.218} C_VEL
LIN {X 0,Y 720.135,Z 610.96,A -85,B 0,C 180,E1 34689.346,E2 34689.346} C_VEL
LIN {X 0,Y 720.154,Z 610.959,A -85,B 0,C 180,E1 34686.857,E2 34686.857} C_VEL
LIN {X 0,Y 720.216,Z 610.951,A -85,B 0,C 180,E1 34683.884,E2 34683.884} C_VEL
LIN {X 0,Y 720.214,Z 610.958,A -85,B 0,C 180,E1 34680.91,E2 34680.91} C_VEL
LIN {X 0,Y 720.218,Z 610.95,A -85,B 0,C 180,E1 34677.834,E2 34677.834} C_VEL
LIN {X 0,Y 720.173,Z 610.959,A -85,B 0,C 180,E1 34674.879,E2 34674.879} C_VEL
LIN {X 0,Y 720.134,Z 610.959,A -85,B 0,C 180,E1 34672.362,E2 34672.362} C_VEL
LIN {X 0,Y 720.208,Z 610.955,A -85,B 0,C 180,E1 34669.464,E2 34669.464} C_VEL
LIN {X 0,Y 720.168,Z 610.956,A -85,B 0,C 180,E1 34666.674,E2 34666.674} C_VEL
LIN {X 0,Y 720.21,Z 610.954,A -85,B 0,C 180,E1 34663.898,E2 34663.898} C_VEL
